LIN{ E6POS: X 741.7167, Y -17.0940, Z -126.0150, A 0, B 90, C 0, E1 0, E2 0, E3 0, E4 0 } C_DIS
LIN{ E6POS: X 740.7177, Y -17.1387, Z -126.0150, A 0, B 90, C 0, E1 0, E2 0, E3 0, E4 0 } C_DIS
LIN{ E6POS: X 739.8800, Y -17.1763, Z -126.0150, A 0, B 90, C 0, E1 0, E2 0, E3 0, E4 0 } C_DIS
LIN{ E6POS: X 739.6024, Y -17.2342, Z -126.0150, A 0, B 90, C 0, E1 0, E2 0, E3 0, E4 0 } C_DIS
LIN{ E6POS: X 738.6175, Y -17.4075, Z -126.0150, A 0, B 90, C 0, E1 0, E2 0, E3 0, E4 0 } C_DIS
LIN{ E6POS: X 737.6326, Y -17.5807, Z -126.0150, A 0, B 90, C 0, E1 0, E2 0, E3 0, E4 0 } C_DIS
LIN{ E6POS: X 736.6477, Y -17.7539, Z -126.0150, A 0, B 90, C 0, E1 0, E2 0, E3 0, E4 0 } C_DIS
LIN{ E6POS: X 736.0951, Y -17.8511, Z -126.0150, A 0, B 90, C 0, E1 0, E2 0, E3 0, E4 0 } C_DIS
LIN{ E6POS: X 736.0012, Y -17.9380, Z -126.0150, A 0, B 90, C 0, E1 0, E2 0, E3 0, E4 0 } C_DIS
LIN{ E6POS: X 735.2228, Y -18.5657, Z -126.0150, A 0, B 90, C 0, E1 0, E2 0, E3 0, E4 0 } C_DIS
LIN{ E6POS: X 734.8225, Y -18.8885, Z -126.0150, A 0, B 90, C 0, E1 0, E2 0, E3 0, E4 0 } C_DIS
LIN{ E6POS: X 735.4953, Y -19.6283, Z -126.0150, A 0, B 90, C 0, E1 0, E2 0, E3 0, E4 0 } C_DIS
LIN{ E6POS: X 735.9742, Y -20.1550, Z -126.0150, A 0, B 90, C 0, E1 0, E2 0, E3 0, E4 0 } C_DIS
LIN{ E6POS: X 736.0644, Y -20.2679, Z -126.0150, A 0, B 90, C 0, E1 0, E2 0, E3 0, E4 0 } C_DIS
LIN{ E6POS: X 736.9769, Y -20.6771, Z -126.0150, A 0, B 90, C 0, E1 0, E2 0, E3 0, E4 0 } C_DIS
LIN{ E6POS: X 737.8893, Y -21.0862, Z -126.0150, A 0, B 90, C 0, E1 0, E2 0, E3 0, E4 0 } C_DIS
LIN{ E6POS: X 738.8018, Y -21.4953, Z -126.0150, A 0, B 90, C 0, E1 0, E2 0, E3 0, E4 0 } C_DIS
LIN{ E6POS: X 739.5476, Y -21.8297, Z -126.0150, A 0, B 90, C 0, E1 0, E2 0, E3 0, E4 0 } C_DIS
LIN{ E6POS: X 739.8221, Y -21.9661, Z -126.0150, A 0, B 90, C 0, E1 0, E2 0, E3 0, E4 0 } C_DIS
LIN{ E6POS: X 740.7757, Y -22.2672, Z -126.0150, A 0, B 90, C 0, E1 0, E2 0, E3 0, E4 0 } C_DIS
LIN{ E6POS: X 741.7293, Y -22.5683, Z -126.0150, A 0, B 90, C 0, E1 0, E2 0, E3 0, E4 0 } C_DIS
LIN{ E6POS: X 742.6829, Y -22.8694, Z -126.0150, A 0, B 90, C 0, E1 0, E2 0, E3 0, E4 0 } C_DIS
LIN{ E6POS: X 743.6365, Y -23.1705, Z -126.0150, A 0, B 90, C 0, E1 0, E2 0, E3 0, E4 0 } C_DIS
LIN{ E6POS: X 744.5901, Y -23.4716, Z -126.0150, A 0, B 90, C 0, E1 0, E2 0, E3 0, E4 0 } C_DIS
LIN{ E6POS: X 745.5437, Y -23.7727, Z -126.0150, A 0, B 90, C 0, E1 0, E2 0, E3 0, E4 0 } C_DIS
LIN{ E6POS: X 745.6394, Y -23.8029, Z -126.0150, A 0, B 90, C 0, E1 0, E2 0, E3 0, E4 0 } C_DIS
LIN{ E6POS: X 746.0988, Y -23.9598, Z -126.0150, A 0, B 90, C 0, E1 0, E2 0, E3 0, E4 0 } C_DIS
LIN{ E6POS: X 747.0681, Y -24.2056, Z -126.0150, A 0, B 90, C 0, E1 0, E2 0, E3 0, E4 0 } C_DIS
LIN{ E6POS: X 748.0375, Y -24.4513, Z -126.0150, A 0, B 90, C 0, E1 0, E2 0, E3 0, E4 0 } C_DIS
LIN{ E6POS: X 749.0068, Y -24.6971, Z -126.0150, A 0, B 90, C 0, E1 0, E2 0, E3 0, E4 0 } C_DIS
LIN{ E6POS: X 749.9761, Y -24.9428, Z -126.0150, A 0, B 90, C 0, E1 0, E2 0, E3 0, E4 0 } C_DIS
LIN{ E6POS: X 750.9455, Y -25.1886, Z -126.0150, A 0, B 90, C 0, E1 0, E2 0, E3 0, E4 0 } C_DIS
LIN{ E6POS: X 751.9148, Y -25.4344, Z -126.0150, A 0, B 90, C 0, E1 0, E2 0, E3 0, E4 0 } C_DIS
LIN{ E6POS: X 752.8841, Y -25.6801, Z -126.0150, A 0, B 90, C 0, E1 0, E2 0, E3 0, E4 0 } C_DIS
LIN{ E6POS: X 753.3483, Y -25.7978, Z -126.0150, A 0, B 90, C 0, E1 0, E2 0, E3 0, E4 0 } C_DIS
LIN{ E6POS: X 753.9231, Y -25.9528, Z -126.0150, A 0, B 90, C 0, E1 0, E2 0, E3 0, E4 0 } C_DIS
LIN{ E6POS: X 754.9035, Y -26.1500, Z -126.0150, A 0, B 90, C 0, E1 0, E2 0, E3 0, E4 0 } C_DIS
LIN{ E6POS: X 755.8838, Y -26.3472, Z -126.0150, A 0, B 90, C 0, E1 0, E2 0, E3 0, E4 0 } C_DIS
LIN{ E6POS: X 756.8642, Y -26.5444, Z -126.0150, A 0, B 90, C 0, E1 0, E2 0, E3 0, E4 0 } C_DIS
LIN{ E6POS: X 757.8446, Y -26.7416, Z -126.0150, A 0, B 90, C 0, E1 0, E2 0, E3 0, E4 0 } C_DIS
LIN{ E6POS: X 758.8249, Y -26.9388, Z -126.0150, A 0, B 90, C 0, E1 0, E2 0, E3 0, E4 0 } C_DIS
LIN{ E6POS: X 759.8053, Y -27.1360, Z -126.0150, A 0, B 90, C 0, E1 0, E2 0, E3 0, E4 0 } C_DIS
LIN{ E6POS: X 760.7857, Y -27.3332, Z -126.0150, A 0, B 90, C 0, E1 0, E2 0, E3 0, E4 0 } C_DIS
LIN{ E6POS: X 761.7005, Y -27.5172, Z -126.0150, A 0, B 90, C 0, E1 0, E2 0, E3 0, E4 0 } C_DIS
LIN{ E6POS: X 762.3215, Y -27.6477, Z -126.0150, A 0, B 90, C 0, E1 0, E2 0, E3 0, E4 0 } C_DIS
LIN{ E6POS: X 763.3122, Y -27.7837, Z -126.0150, A 0, B 90, C 0, E1 0, E2 0, E3 0, E4 0 } C_DIS
LIN{ E6POS: X 764.3029, Y -27.9196, Z -126.0150, A 0, B 90, C 0, E1 0, E2 0, E3 0, E4 0 } C_DIS
LIN{ E6POS: X 765.2937, Y -28.0556, Z -126.0150, A 0, B 90, C 0, E1 0, E2 0, E3 0, E4 0 } C_DIS
LIN{ E6POS: X 766.2844, Y -28.1916, Z -126.0150, A 0, B 90, C 0, E1 0, E2 0, E3 0, E4 0 } C_DIS
LIN{ E6POS: X 767.2751, Y -28.3276, Z -126.0150, A 0, B 90, C 0, E1 0, E2 0, E3 0, E4 0 } C_DIS
LIN{ E6POS: X 768.2658, Y -28.4636, Z -126.0150, A 0, B 90, C 0, E1 0, E2 0, E3 0, E4 0 } C_DIS
LIN{ E6POS: X 769.2565, Y -28.5995, Z -126.0150, A 0, B 90, C 0, E1 0, E2 0, E3 0, E4 0 } C_DIS
LIN{ E6POS: X 769.7261, Y -28.6640, Z -126.0150, A 0, B 90, C 0, E1 0, E2 0, E3 0, E4 0 } C_DIS
LIN{ E6POS: X 770.3238, Y -28.7475, Z -126.0150, A 0, B 90, C 0, E1 0, E2 0, E3 0, E4 0 } C_DIS
LIN{ E6POS: X 771.3233, Y -28.7792, Z -126.0150, A 0, B 90, C 0, E1 0, E2 0, E3 0, E4 0 } C_DIS
LIN{ E6POS: X 772.3228, Y -28.8109, Z -126.0150, A 0, B 90, C 0, E1 0, E2 0, E3 0, E4 0 } C_DIS
LIN{ E6POS: X 773.3223, Y -28.8426, Z -126.0150, A 0, B 90, C 0, E1 0, E2 0, E3 0, E4 0 } C_DIS
LIN{ E6POS: X 774.3218, Y -28.8743, Z -126.0150, A 0, B 90, C 0, E1 0, E2 0, E3 0, E4 0 } C_DIS
LIN{ E6POS: X 775.3213, Y -28.9060, Z -126.0150, A 0, B 90, C 0, E1 0, E2 0, E3 0, E4 0 } C_DIS
LIN{ E6POS: X 776.3208, Y -28.9377, Z -126.0150, A 0, B 90, C 0, E1 0, E2 0, E3 0, E4 0 } C_DIS
LIN{ E6POS: X 776.4510, Y -28.9418, Z -126.0150, A 0, B 90, C 0, E1 0, E2 0, E3 0, E4 0 } C_DIS
LIN{ E6POS: X 776.9561, Y -28.9557, Z -126.0150, A 0, B 90, C 0, E1 0, E2 0, E3 0, E4 0 } C_DIS
LIN{ E6POS: X 777.9387, Y -29.1413, Z -126.0150, A 0, B 90, C 0, E1 0, E2 0, E3 0, E4 0 } C_DIS
LIN{ E6POS: X 778.9214, Y -29.3269, Z -126.0150, A 0, B 90, C 0, E1 0, E2 0, E3 0, E4 0 } C_DIS
LIN{ E6POS: X 779.9040, Y -29.5125, Z -126.0150, A 0, B 90, C 0, E1 0, E2 0, E3 0, E4 0 } C_DIS
LIN{ E6POS: X 780.8866, Y -29.6981, Z -126.0150, A 0, B 90, C 0, E1 0, E2 0, E3 0, E4 0 } C_DIS
LIN{ E6POS: X 781.5842, Y -29.8299, Z -126.0150, A 0, B 90, C 0, E1 0, E2 0, E3 0, E4 0 } C_DIS
LIN{ E6POS: X 781.9729, Y -29.9044, Z -126.0150, A 0, B 90, C 0, E1 0, E2 0, E3 0, E4 0 } C_DIS
LIN{ E6POS: X 782.6620, Y -30.6291, Z -126.0150, A 0, B 90, C 0, E1 0, E2 0, E3 0, E4 0 } C_DIS
LIN{ E6POS: X 783.3511, Y -31.3537, Z -126.0150, A 0, B 90, C 0, E1 0, E2 0, E3 0, E4 0 } C_DIS
LIN{ E6POS: X 784.0403, Y -32.0783, Z -126.0150, A 0, B 90, C 0, E1 0, E2 0, E3 0, E4 0 } C_DIS
LIN{ E6POS: X 784.7294, Y -32.8030, Z -126.0150, A 0, B 90, C 0, E1 0, E2 0, E3 0, E4 0 } C_DIS
LIN{ E6POS: X 784.8800, Y -32.9613, Z -126.0150, A 0, B 90, C 0, E1 0, E2 0, E3 0, E4 0 } C_DIS
LIN{ E6POS: X 785.1281, Y -33.2266, Z -126.0150, A 0, B 90, C 0, E1 0, E2 0, E3 0, E4 0 } C_DIS
LIN{ E6POS: X 785.2695, Y -34.2166, Z -126.0150, A 0, B 90, C 0, E1 0, E2 0, E3 0, E4 0 } C_DIS
LIN{ E6POS: X 785.4109, Y -35.2065, Z -126.0150, A 0, B 90, C 0, E1 0, E2 0, E3 0, E4 0 } C_DIS
LIN{ E6POS: X 785.5523, Y -36.1965, Z -126.0150, A 0, B 90, C 0, E1 0, E2 0, E3 0, E4 0 } C_DIS
LIN{ E6POS: X 785.6937, Y -37.1864, Z -126.0150, A 0, B 90, C 0, E1 0, E2 0, E3 0, E4 0 } C_DIS
LIN{ E6POS: X 785.8351, Y -38.1764, Z -126.0150, A 0, B 90, C 0, E1 0, E2 0, E3 0, E4 0 } C_DIS
LIN{ E6POS: X 785.9765, Y -39.1663, Z -126.0150, A 0, B 90, C 0, E1 0, E2 0, E3 0, E4 0 } C_DIS
LIN{ E6POS: X 786.0909, Y -39.9674, Z -126.0150, A 0, B 90, C 0, E1 0, E2 0, E3 0, E4 0 } C_DIS
LIN{ E6POS: X 786.1747, Y -40.5536, Z -126.0150, A 0, B 90, C 0, E1 0, E2 0, E3 0, E4 0 } C_DIS
LIN{ E6POS: X 786.0743, Y -41.5485, Z -126.0150, A 0, B 90, C 0, E1 0, E2 0, E3 0, E4 0 } C_DIS
LIN{ E6POS: X 785.9740, Y -42.5435, Z -126.0150, A 0, B 90, C 0, E1 0, E2 0, E3 0, E4 0 } C_DIS
LIN{ E6POS: X 785.8737, Y -43.5384, Z -126.0150, A 0, B 90, C 0, E1 0, E2 0, E3 0, E4 0 } C_DIS
LIN{ E6POS: X 785.7734, Y -44.5334, Z -126.0150, A 0, B 90, C 0, E1 0, E2 0, E3 0, E4 0 } C_DIS
LIN{ E6POS: X 785.6731, Y -45.5283, Z -126.0150, A 0, B 90, C 0, E1 0, E2 0, E3 0, E4 0 } C_DIS
LIN{ E6POS: X 785.5728, Y -46.5233, Z -126.0150, A 0, B 90, C 0, E1 0, E2 0, E3 0, E4 0 } C_DIS
LIN{ E6POS: X 785.4725, Y -47.5183, Z -126.0150, A 0, B 90, C 0, E1 0, E2 0, E3 0, E4 0 } C_DIS
LIN{ E6POS: X 785.3721, Y -48.5132, Z -126.0150, A 0, B 90, C 0, E1 0, E2 0, E3 0, E4 0 } C_DIS
LIN{ E6POS: X 785.2718, Y -49.5082, Z -126.0150, A 0, B 90, C 0, E1 0, E2 0, E3 0, E4 0 } C_DIS
LIN{ E6POS: X 785.1715, Y -50.5031, Z -126.0150, A 0, B 90, C 0, E1 0, E2 0, E3 0, E4 0 } C_DIS
LIN{ E6POS: X 785.0712, Y -51.4981, Z -126.0150, A 0, B 90, C 0, E1 0, E2 0, E3 0, E4 0 } C_DIS
LIN{ E6POS: X 784.9721, Y -52.4813, Z -126.0150, A 0, B 90, C 0, E1 0, E2 0, E3 0, E4 0 } C_DIS
LIN{ E6POS: X 784.8718, Y -53.4762, Z -126.0150, A 0, B 90, C 0, E1 0, E2 0, E3 0, E4 0 } C_DIS
LIN{ E6POS: X 784.8675, Y -53.5185, Z -126.0150, A 0, B 90, C 0, E1 0, E2 0, E3 0, E4 0 } C_DIS
LIN{ E6POS: X 784.6915, Y -54.5029, Z -126.0150, A 0, B 90, C 0, E1 0, E2 0, E3 0, E4 0 } C_DIS
LIN{ E6POS: X 784.5156, Y -55.4873, Z -126.0150, A 0, B 90, C 0, E1 0, E2 0, E3 0, E4 0 } C_DIS
LIN{ E6POS: X 784.3396, Y -56.4717, Z -126.0150, A 0, B 90, C 0, E1 0, E2 0, E3 0, E4 0 } C_DIS
LIN{ E6POS: X 784.1637, Y -57.4560, Z -126.0150, A 0, B 90, C 0, E1 0, E2 0, E3 0, E4 0 } C_DIS
LIN{ E6POS: X 783.9877, Y -58.4404, Z -126.0150, A 0, B 90, C 0, E1 0, E2 0, E3 0, E4 0 } C_DIS
LIN{ E6POS: X 783.8118, Y -59.4248, Z -126.0150, A 0, B 90, C 0, E1 0, E2 0, E3 0, E4 0 } C_DIS
LIN{ E6POS: X 783.6358, Y -60.4092, Z -126.0150, A 0, B 90, C 0, E1 0, E2 0, E3 0, E4 0 } C_DIS
LIN{ E6POS: X 783.4599, Y -61.3936, Z -126.0150, A 0, B 90, C 0, E1 0, E2 0, E3 0, E4 0 } C_DIS
LIN{ E6POS: X 783.2839, Y -62.3780, Z -126.0150, A 0, B 90, C 0, E1 0, E2 0, E3 0, E4 0 } C_DIS
LIN{ E6POS: X 783.1080, Y -63.3624, Z -126.0150, A 0, B 90, C 0, E1 0, E2 0, E3 0, E4 0 } C_DIS
LIN{ E6POS: X 782.9320, Y -64.3468, Z -126.0150, A 0, B 90, C 0, E1 0, E2 0, E3 0, E4 0 } C_DIS
LIN{ E6POS: X 782.7561, Y -65.3312, Z -126.0150, A 0, B 90, C 0, E1 0, E2 0, E3 0, E4 0 } C_DIS
LIN{ E6POS: X 782.5801, Y -66.3156, Z -126.0150, A 0, B 90, C 0, E1 0, E2 0, E3 0, E4 0 } C_DIS
LIN{ E6POS: X 782.4042, Y -67.3000, Z -126.0150, A 0, B 90, C 0, E1 0, E2 0, E3 0, E4 0 } C_DIS
LIN{ E6POS: X 782.2282, Y -68.2844, Z -126.0150, A 0, B 90, C 0, E1 0, E2 0, E3 0, E4 0 } C_DIS
LIN{ E6POS: X 782.0523, Y -69.2688, Z -126.0150, A 0, B 90, C 0, E1 0, E2 0, E3 0, E4 0 } C_DIS
LIN{ E6POS: X 782.0402, Y -69.3364, Z -126.0150, A 0, B 90, C 0, E1 0, E2 0, E3 0, E4 0 } C_DIS
LIN{ E6POS: X 781.8642, Y -70.3208, Z -126.0150, A 0, B 90, C 0, E1 0, E2 0, E3 0, E4 0 } C_DIS
LIN{ E6POS: X 781.7943, Y -70.7119, Z -126.0150, A 0, B 90, C 0, E1 0, E2 0, E3 0, E4 0 } C_DIS
LIN{ E6POS: X 781.5865, Y -71.6900, Z -126.0150, A 0, B 90, C 0, E1 0, E2 0, E3 0, E4 0 } C_DIS
LIN{ E6POS: X 781.3787, Y -72.6682, Z -126.0150, A 0, B 90, C 0, E1 0, E2 0, E3 0, E4 0 } C_DIS
LIN{ E6POS: X 781.1709, Y -73.6464, Z -126.0150, A 0, B 90, C 0, E1 0, E2 0, E3 0, E4 0 } C_DIS
LIN{ E6POS: X 780.9631, Y -74.6245, Z -126.0150, A 0, B 90, C 0, E1 0, E2 0, E3 0, E4 0 } C_DIS
LIN{ E6POS: X 780.7553, Y -75.6027, Z -126.0150, A 0, B 90, C 0, E1 0, E2 0, E3 0, E4 0 } C_DIS
LIN{ E6POS: X 780.5475, Y -76.5809, Z -126.0150, A 0, B 90, C 0, E1 0, E2 0, E3 0, E4 0 } C_DIS
LIN{ E6POS: X 780.3397, Y -77.5590, Z -126.0150, A 0, B 90, C 0, E1 0, E2 0, E3 0, E4 0 } C_DIS
LIN{ E6POS: X 780.1319, Y -78.5372, Z -126.0150, A 0, B 90, C 0, E1 0, E2 0, E3 0, E4 0 } C_DIS
LIN{ E6POS: X 779.9241, Y -79.5154, Z -126.0150, A 0, B 90, C 0, E1 0, E2 0, E3 0, E4 0 } C_DIS
LIN{ E6POS: X 779.7163, Y -80.4936, Z -126.0150, A 0, B 90, C 0, E1 0, E2 0, E3 0, E4 0 } C_DIS
LIN{ E6POS: X 779.5085, Y -81.4717, Z -126.0150, A 0, B 90, C 0, E1 0, E2 0, E3 0, E4 0 } C_DIS
LIN{ E6POS: X 779.3007, Y -82.4499, Z -126.0150, A 0, B 90, C 0, E1 0, E2 0, E3 0, E4 0 } C_DIS
LIN{ E6POS: X 779.0929, Y -83.4281, Z -126.0150, A 0, B 90, C 0, E1 0, E2 0, E3 0, E4 0 } C_DIS
LIN{ E6POS: X 778.8851, Y -84.4062, Z -126.0150, A 0, B 90, C 0, E1 0, E2 0, E3 0, E4 0 } C_DIS
LIN{ E6POS: X 778.6773, Y -85.3844, Z -126.0150, A 0, B 90, C 0, E1 0, E2 0, E3 0, E4 0 } C_DIS
LIN{ E6POS: X 778.4695, Y -86.3626, Z -126.0150, A 0, B 90, C 0, E1 0, E2 0, E3 0, E4 0 } C_DIS
LIN{ E6POS: X 778.2617, Y -87.3408, Z -126.0150, A 0, B 90, C 0, E1 0, E2 0, E3 0, E4 0 } C_DIS
LIN{ E6POS: X 778.0539, Y -88.3189, Z -126.0150, A 0, B 90, C 0, E1 0, E2 0, E3 0, E4 0 } C_DIS
LIN{ E6POS: X 777.8830, Y -89.1233, Z -126.0150, A 0, B 90, C 0, E1 0, E2 0, E3 0, E4 0 } C_DIS
LIN{ E6POS: X 777.6752, Y -90.1015, Z -126.0150, A 0, B 90, C 0, E1 0, E2 0, E3 0, E4 0 } C_DIS
LIN{ E6POS: X 777.5429, Y -90.7243, Z -126.0150, A 0, B 90, C 0, E1 0, E2 0, E3 0, E4 0 } C_DIS
LIN{ E6POS: X 777.3226, Y -91.6997, Z -126.0150, A 0, B 90, C 0, E1 0, E2 0, E3 0, E4 0 } C_DIS
LIN{ E6POS: X 777.1022, Y -92.6751, Z -126.0150, A 0, B 90, C 0, E1 0, E2 0, E3 0, E4 0 } C_DIS
LIN{ E6POS: X 776.8819, Y -93.6506, Z -126.0150, A 0, B 90, C 0, E1 0, E2 0, E3 0, E4 0 } C_DIS
LIN{ E6POS: X 776.6615, Y -94.6260, Z -126.0150, A 0, B 90, C 0, E1 0, E2 0, E3 0, E4 0 } C_DIS
LIN{ E6POS: X 776.4412, Y -95.6014, Z -126.0150, A 0, B 90, C 0, E1 0, E2 0, E3 0, E4 0 } C_DIS
LIN{ E6POS: X 776.2208, Y -96.5768, Z -126.0150, A 0, B 90, C 0, E1 0, E2 0, E3 0, E4 0 } C_DIS
LIN{ E6POS: X 776.0005, Y -97.5522, Z -126.0150, A 0, B 90, C 0, E1 0, E2 0, E3 0, E4 0 } C_DIS
LIN{ E6POS: X 775.7802, Y -98.5277, Z -126.0150, A 0, B 90, C 0, E1 0, E2 0, E3 0, E4 0 } C_DIS
LIN{ E6POS: X 775.5598, Y -99.5031, Z -126.0150, A 0, B 90, C 0, E1 0, E2 0, E3 0, E4 0 } C_DIS
LIN{ E6POS: X 775.3395, Y -100.4785, Z -126.0150, A 0, B 90, C 0, E1 0, E2 0, E3 0, E4 0 } C_DIS
LIN{ E6POS: X 775.1191, Y -101.4539, Z -126.0150, A 0, B 90, C 0, E1 0, E2 0, E3 0, E4 0 } C_DIS
LIN{ E6POS: X 774.8988, Y -102.4294, Z -126.0150, A 0, B 90, C 0, E1 0, E2 0, E3 0, E4 0 } C_DIS
LIN{ E6POS: X 774.6784, Y -103.4048, Z -126.0150, A 0, B 90, C 0, E1 0, E2 0, E3 0, E4 0 } C_DIS
LIN{ E6POS: X 774.4581, Y -104.3802, Z -126.0150, A 0, B 90, C 0, E1 0, E2 0, E3 0, E4 0 } C_DIS
LIN{ E6POS: X 774.2377, Y -105.3556, Z -126.0150, A 0, B 90, C 0, E1 0, E2 0, E3 0, E4 0 } C_DIS
LIN{ E6POS: X 774.0174, Y -106.3310, Z -126.0150, A 0, B 90, C 0, E1 0, E2 0, E3 0, E4 0 } C_DIS
LIN{ E6POS: X 773.7970, Y -107.3065, Z -126.0150, A 0, B 90, C 0, E1 0, E2 0, E3 0, E4 0 } C_DIS
LIN{ E6POS: X 773.5767, Y -108.2819, Z -126.0150, A 0, B 90, C 0, E1 0, E2 0, E3 0, E4 0 } C_DIS
LIN{ E6POS: X 773.3564, Y -109.2573, Z -126.0150, A 0, B 90, C 0, E1 0, E2 0, E3 0, E4 0 } C_DIS
LIN{ E6POS: X 773.1360, Y -110.2327, Z -126.0150, A 0, B 90, C 0, E1 0, E2 0, E3 0, E4 0 } C_DIS
LIN{ E6POS: X 773.0909, Y -110.4324, Z -126.0150, A 0, B 90, C 0, E1 0, E2 0, E3 0, E4 0 } C_DIS
LIN{ E6POS: X 772.8706, Y -111.4079, Z -126.0150, A 0, B 90, C 0, E1 0, E2 0, E3 0, E4 0 } C_DIS
LIN{ E6POS: X 772.7038, Y -112.1462, Z -126.0150, A 0, B 90, C 0, E1 0, E2 0, E3 0, E4 0 } C_DIS
LIN{ E6POS: X 772.0412, Y -111.3972, Z -126.0150, A 0, B 90, C 0, E1 0, E2 0, E3 0, E4 0 } C_DIS
LIN{ E6POS: X 771.3787, Y -110.6481, Z -126.0150, A 0, B 90, C 0, E1 0, E2 0, E3 0, E4 0 } C_DIS
LIN{ E6POS: X 770.7162, Y -109.8991, Z -126.0150, A 0, B 90, C 0, E1 0, E2 0, E3 0, E4 0 } C_DIS
LIN{ E6POS: X 770.2453, Y -109.3667, Z -126.0150, A 0, B 90, C 0, E1 0, E2 0, E3 0, E4 0 } C_DIS
LIN{ E6POS: X 770.0315, Y -109.1250, Z -126.0150, A 0, B 90, C 0, E1 0, E2 0, E3 0, E4 0 } C_DIS
LIN{ E6POS: X 769.2905, Y -108.4535, Z -126.0150, A 0, B 90, C 0, E1 0, E2 0, E3 0, E4 0 } C_DIS
LIN{ E6POS: X 768.5495, Y -107.7819, Z -126.0150, A 0, B 90, C 0, E1 0, E2 0, E3 0, E4 0 } C_DIS
LIN{ E6POS: X 767.8086, Y -107.1104, Z -126.0150, A 0, B 90, C 0, E1 0, E2 0, E3 0, E4 0 } C_DIS
LIN{ E6POS: X 767.0676, Y -106.4389, Z -126.0150, A 0, B 90, C 0, E1 0, E2 0, E3 0, E4 0 } C_DIS
LIN{ E6POS: X 766.8332, Y -106.2265, Z -126.0150, A 0, B 90, C 0, E1 0, E2 0, E3 0, E4 0 } C_DIS
LIN{ E6POS: X 766.5571, Y -105.9757, Z -126.0150, A 0, B 90, C 0, E1 0, E2 0, E3 0, E4 0 } C_DIS
LIN{ E6POS: X 766.1563, Y -105.7065, Z -126.0150, A 0, B 90, C 0, E1 0, E2 0, E3 0, E4 0 } C_DIS
LIN{ E6POS: X 765.3256, Y -105.1498, Z -126.0150, A 0, B 90, C 0, E1 0, E2 0, E3 0, E4 0 } C_DIS
LIN{ E6POS: X 764.4949, Y -104.5931, Z -126.0150, A 0, B 90, C 0, E1 0, E2 0, E3 0, E4 0 } C_DIS
LIN{ E6POS: X 763.6642, Y -104.0363, Z -126.0150, A 0, B 90, C 0, E1 0, E2 0, E3 0, E4 0 } C_DIS
LIN{ E6POS: X 762.8335, Y -103.4796, Z -126.0150, A 0, B 90, C 0, E1 0, E2 0, E3 0, E4 0 } C_DIS
LIN{ E6POS: X 762.0028, Y -102.9229, Z -126.0150, A 0, B 90, C 0, E1 0, E2 0, E3 0, E4 0 } C_DIS
LIN{ E6POS: X 761.4803, Y -102.5727, Z -126.0150, A 0, B 90, C 0, E1 0, E2 0, E3 0, E4 0 } C_DIS
LIN{ E6POS: X 760.8926, Y -102.2760, Z -126.0150, A 0, B 90, C 0, E1 0, E2 0, E3 0, E4 0 } C_DIS
LIN{ E6POS: X 760.0004, Y -101.8244, Z -126.0150, A 0, B 90, C 0, E1 0, E2 0, E3 0, E4 0 } C_DIS
LIN{ E6POS: X 759.1082, Y -101.3728, Z -126.0150, A 0, B 90, C 0, E1 0, E2 0, E3 0, E4 0 } C_DIS
LIN{ E6POS: X 758.2159, Y -100.9213, Z -126.0150, A 0, B 90, C 0, E1 0, E2 0, E3 0, E4 0 } C_DIS
LIN{ E6POS: X 757.3237, Y -100.4697, Z -126.0150, A 0, B 90, C 0, E1 0, E2 0, E3 0, E4 0 } C_DIS
LIN{ E6POS: X 756.4315, Y -100.0181, Z -126.0150, A 0, B 90, C 0, E1 0, E2 0, E3 0, E4 0 } C_DIS
LIN{ E6POS: X 755.5392, Y -99.5665, Z -126.0150, A 0, B 90, C 0, E1 0, E2 0, E3 0, E4 0 } C_DIS
LIN{ E6POS: X 754.6470, Y -99.1150, Z -126.0150, A 0, B 90, C 0, E1 0, E2 0, E3 0, E4 0 } C_DIS
LIN{ E6POS: X 753.9986, Y -98.7868, Z -126.0150, A 0, B 90, C 0, E1 0, E2 0, E3 0, E4 0 } C_DIS
LIN{ E6POS: X 753.1615, Y -98.4535, Z -126.0150, A 0, B 90, C 0, E1 0, E2 0, E3 0, E4 0 } C_DIS
LIN{ E6POS: X 752.2338, Y -98.0803, Z -126.0150, A 0, B 90, C 0, E1 0, E2 0, E3 0, E4 0 } C_DIS
LIN{ E6POS: X 751.3060, Y -97.7070, Z -126.0150, A 0, B 90, C 0, E1 0, E2 0, E3 0, E4 0 } C_DIS
LIN{ E6POS: X 750.3783, Y -97.3338, Z -126.0150, A 0, B 90, C 0, E1 0, E2 0, E3 0, E4 0 } C_DIS
LIN{ E6POS: X 749.4506, Y -96.9605, Z -126.0150, A 0, B 90, C 0, E1 0, E2 0, E3 0, E4 0 } C_DIS
LIN{ E6POS: X 748.5228, Y -96.5873, Z -126.0150, A 0, B 90, C 0, E1 0, E2 0, E3 0, E4 0 } C_DIS
LIN{ E6POS: X 747.5951, Y -96.2140, Z -126.0150, A 0, B 90, C 0, E1 0, E2 0, E3 0, E4 0 } C_DIS
LIN{ E6POS: X 746.6674, Y -95.8408, Z -126.0150, A 0, B 90, C 0, E1 0, E2 0, E3 0, E4 0 } C_DIS
LIN{ E6POS: X 745.7396, Y -95.4675, Z -126.0150, A 0, B 90, C 0, E1 0, E2 0, E3 0, E4 0 } C_DIS
LIN{ E6POS: X 744.8119, Y -95.0943, Z -126.0150, A 0, B 90, C 0, E1 0, E2 0, E3 0, E4 0 } C_DIS
LIN{ E6POS: X 743.8842, Y -94.7210, Z -126.0150, A 0, B 90, C 0, E1 0, E2 0, E3 0, E4 0 } C_DIS
LIN{ E6POS: X 743.3112, Y -94.4905, Z -126.0150, A 0, B 90, C 0, E1 0, E2 0, E3 0, E4 0 } C_DIS
LIN{ E6POS: X 742.3695, Y -94.1539, Z -126.0150, A 0, B 90, C 0, E1 0, E2 0, E3 0, E4 0 } C_DIS
LIN{ E6POS: X 742.3638, Y -94.1519, Z -126.0150, A 0, B 90, C 0, E1 0, E2 0, E3 0, E4 0 } C_DIS
LIN{ E6POS: X 741.4234, Y -93.8116, Z -126.0150, A 0, B 90, C 0, E1 0, E2 0, E3 0, E4 0 } C_DIS
LIN{ E6POS: X 740.4831, Y -93.4714, Z -126.0150, A 0, B 90, C 0, E1 0, E2 0, E3 0, E4 0 } C_DIS
LIN{ E6POS: X 739.5428, Y -93.1311, Z -126.0150, A 0, B 90, C 0, E1 0, E2 0, E3 0, E4 0 } C_DIS
LIN{ E6POS: X 738.6024, Y -92.7908, Z -126.0150, A 0, B 90, C 0, E1 0, E2 0, E3 0, E4 0 } C_DIS
LIN{ E6POS: X 737.6621, Y -92.4506, Z -126.0150, A 0, B 90, C 0, E1 0, E2 0, E3 0, E4 0 } C_DIS
LIN{ E6POS: X 736.7218, Y -92.1103, Z -126.0150, A 0, B 90, C 0, E1 0, E2 0, E3 0, E4 0 } C_DIS
LIN{ E6POS: X 735.7814, Y -91.7701, Z -126.0150, A 0, B 90, C 0, E1 0, E2 0, E3 0, E4 0 } C_DIS
LIN{ E6POS: X 734.8411, Y -91.4298, Z -126.0150, A 0, B 90, C 0, E1 0, E2 0, E3 0, E4 0 } C_DIS
LIN{ E6POS: X 733.9008, Y -91.0896, Z -126.0150, A 0, B 90, C 0, E1 0, E2 0, E3 0, E4 0 } C_DIS
LIN{ E6POS: X 732.9604, Y -90.7493, Z -126.0150, A 0, B 90, C 0, E1 0, E2 0, E3 0, E4 0 } C_DIS
LIN{ E6POS: X 732.0201, Y -90.4091, Z -126.0150, A 0, B 90, C 0, E1 0, E2 0, E3 0, E4 0 } C_DIS
LIN{ E6POS: X 731.1955, Y -90.1107, Z -126.0150, A 0, B 90, C 0, E1 0, E2 0, E3 0, E4 0 } C_DIS
LIN{ E6POS: X 730.2766, Y -89.7980, Z -126.0150, A 0, B 90, C 0, E1 0, E2 0, E3 0, E4 0 } C_DIS
LIN{ E6POS: X 729.3309, Y -89.4731, Z -126.0150, A 0, B 90, C 0, E1 0, E2 0, E3 0, E4 0 } C_DIS
LIN{ E6POS: X 728.3851, Y -89.1482, Z -126.0150, A 0, B 90, C 0, E1 0, E2 0, E3 0, E4 0 } C_DIS
LIN{ E6POS: X 727.4394, Y -88.8233, Z -126.0150, A 0, B 90, C 0, E1 0, E2 0, E3 0, E4 0 } C_DIS
LIN{ E6POS: X 726.4936, Y -88.4984, Z -126.0150, A 0, B 90, C 0, E1 0, E2 0, E3 0, E4 0 } C_DIS
LIN{ E6POS: X 725.5479, Y -88.1735, Z -126.0150, A 0, B 90, C 0, E1 0, E2 0, E3 0, E4 0 } C_DIS
LIN{ E6POS: X 724.6021, Y -87.8486, Z -126.0150, A 0, B 90, C 0, E1 0, E2 0, E3 0, E4 0 } C_DIS
LIN{ E6POS: X 723.6564, Y -87.5237, Z -126.0150, A 0, B 90, C 0, E1 0, E2 0, E3 0, E4 0 } C_DIS
LIN{ E6POS: X 722.7106, Y -87.1988, Z -126.0150, A 0, B 90, C 0, E1 0, E2 0, E3 0, E4 0 } C_DIS
LIN{ E6POS: X 721.7649, Y -86.8739, Z -126.0150, A 0, B 90, C 0, E1 0, E2 0, E3 0, E4 0 } C_DIS
LIN{ E6POS: X 720.8191, Y -86.5490, Z -126.0150, A 0, B 90, C 0, E1 0, E2 0, E3 0, E4 0 } C_DIS
LIN{ E6POS: X 719.8734, Y -86.2242, Z -126.0150, A 0, B 90, C 0, E1 0, E2 0, E3 0, E4 0 } C_DIS
LIN{ E6POS: X 719.4295, Y -86.0717, Z -126.0150, A 0, B 90, C 0, E1 0, E2 0, E3 0, E4 0 } C_DIS
LIN{ E6POS: X 718.6780, Y -85.8163, Z -126.0150, A 0, B 90, C 0, E1 0, E2 0, E3 0, E4 0 } C_DIS
LIN{ E6POS: X 717.7311, Y -85.4947, Z -126.0150, A 0, B 90, C 0, E1 0, E2 0, E3 0, E4 0 } C_DIS
LIN{ E6POS: X 716.7842, Y -85.1732, Z -126.0150, A 0, B 90, C 0, E1 0, E2 0, E3 0, E4 0 } C_DIS
LIN{ E6POS: X 715.8373, Y -84.8517, Z -126.0150, A 0, B 90, C 0, E1 0, E2 0, E3 0, E4 0 } C_DIS
LIN{ E6POS: X 714.8904, Y -84.5302, Z -126.0150, A 0, B 90, C 0, E1 0, E2 0, E3 0, E4 0 } C_DIS
LIN{ E6POS: X 713.9435, Y -84.2087, Z -126.0150, A 0, B 90, C 0, E1 0, E2 0, E3 0, E4 0 } C_DIS
LIN{ E6POS: X 712.9966, Y -83.8871, Z -126.0150, A 0, B 90, C 0, E1 0, E2 0, E3 0, E4 0 } C_DIS
LIN{ E6POS: X 712.0497, Y -83.5656, Z -126.0150, A 0, B 90, C 0, E1 0, E2 0, E3 0, E4 0 } C_DIS
LIN{ E6POS: X 711.1028, Y -83.2441, Z -126.0150, A 0, B 90, C 0, E1 0, E2 0, E3 0, E4 0 } C_DIS
LIN{ E6POS: X 710.1559, Y -82.9226, Z -126.0150, A 0, B 90, C 0, E1 0, E2 0, E3 0, E4 0 } C_DIS
LIN{ E6POS: X 709.7916, Y -82.7989, Z -126.0150, A 0, B 90, C 0, E1 0, E2 0, E3 0, E4 0 } C_DIS
LIN{ E6POS: X 709.3465, Y -82.6322, Z -126.0150, A 0, B 90, C 0, E1 0, E2 0, E3 0, E4 0 } C_DIS
LIN{ E6POS: X 708.4062, Y -82.2918, Z -126.0150, A 0, B 90, C 0, E1 0, E2 0, E3 0, E4 0 } C_DIS
LIN{ E6POS: X 707.4659, Y -81.9515, Z -126.0150, A 0, B 90, C 0, E1 0, E2 0, E3 0, E4 0 } C_DIS
LIN{ E6POS: X 706.5256, Y -81.6111, Z -126.0150, A 0, B 90, C 0, E1 0, E2 0, E3 0, E4 0 } C_DIS
LIN{ E6POS: X 705.5853, Y -81.2708, Z -126.0150, A 0, B 90, C 0, E1 0, E2 0, E3 0, E4 0 } C_DIS
LIN{ E6POS: X 704.6450, Y -80.9305, Z -126.0150, A 0, B 90, C 0, E1 0, E2 0, E3 0, E4 0 } C_DIS
LIN{ E6POS: X 704.0586, Y -80.7182, Z -126.0150, A 0, B 90, C 0, E1 0, E2 0, E3 0, E4 0 } C_DIS
LIN{ E6POS: X 703.8433, Y -80.6180, Z -126.0150, A 0, B 90, C 0, E1 0, E2 0, E3 0, E4 0 } C_DIS
LIN{ E6POS: X 702.9212, Y -80.2310, Z -126.0150, A 0, B 90, C 0, E1 0, E2 0, E3 0, E4 0 } C_DIS
LIN{ E6POS: X 701.9991, Y -79.8440, Z -126.0150, A 0, B 90, C 0, E1 0, E2 0, E3 0, E4 0 } C_DIS
LIN{ E6POS: X 701.2543, Y -79.5315, Z -126.0150, A 0, B 90, C 0, E1 0, E2 0, E3 0, E4 0 } C_DIS
LIN{ E6POS: X 701.2019, Y -79.4530, Z -126.0150, A 0, B 90, C 0, E1 0, E2 0, E3 0, E4 0 } C_DIS
LIN{ E6POS: X 700.4916, Y -78.7491, Z -126.0150, A 0, B 90, C 0, E1 0, E2 0, E3 0, E4 0 } C_DIS
LIN{ E6POS: X 700.4879, Y -78.7454, Z -126.0150, A 0, B 90, C 0, E1 0, E2 0, E3 0, E4 0 } C_DIS
LIN{ E6POS: X 700.7255, Y -77.7740, Z -126.0150, A 0, B 90, C 0, E1 0, E2 0, E3 0, E4 0 } C_DIS
LIN{ E6POS: X 700.8261, Y -77.3633, Z -126.0150, A 0, B 90, C 0, E1 0, E2 0, E3 0, E4 0 } C_DIS
LIN{ E6POS: X 700.8626, Y -77.2328, Z -126.0150, A 0, B 90, C 0, E1 0, E2 0, E3 0, E4 0 } C_DIS
LIN{ E6POS: X 701.0928, Y -76.2597, Z -126.0150, A 0, B 90, C 0, E1 0, E2 0, E3 0, E4 0 } C_DIS
LIN{ E6POS: X 701.1686, Y -75.9391, Z -126.0150, A 0, B 90, C 0, E1 0, E2 0, E3 0, E4 0 } C_DIS
LIN{ E6POS: X 701.2004, Y -75.8212, Z -126.0150, A 0, B 90, C 0, E1 0, E2 0, E3 0, E4 0 } C_DIS
LIN{ E6POS: X 701.4360, Y -74.8493, Z -126.0150, A 0, B 90, C 0, E1 0, E2 0, E3 0, E4 0 } C_DIS
LIN{ E6POS: X 701.5128, Y -74.5323, Z -126.0150, A 0, B 90, C 0, E1 0, E2 0, E3 0, E4 0 } C_DIS
LIN{ E6POS: X 701.5447, Y -74.4166, Z -126.0150, A 0, B 90, C 0, E1 0, E2 0, E3 0, E4 0 } C_DIS
LIN{ E6POS: X 701.7895, Y -73.4470, Z -126.0150, A 0, B 90, C 0, E1 0, E2 0, E3 0, E4 0 } C_DIS
LIN{ E6POS: X 701.8681, Y -73.1360, Z -126.0150, A 0, B 90, C 0, E1 0, E2 0, E3 0, E4 0 } C_DIS
LIN{ E6POS: X 701.9001, Y -73.0237, Z -126.0150, A 0, B 90, C 0, E1 0, E2 0, E3 0, E4 0 } C_DIS
LIN{ E6POS: X 702.1561, Y -72.0570, Z -126.0150, A 0, B 90, C 0, E1 0, E2 0, E3 0, E4 0 } C_DIS
LIN{ E6POS: X 702.2370, Y -71.7511, Z -126.0150, A 0, B 90, C 0, E1 0, E2 0, E3 0, E4 0 } C_DIS
LIN{ E6POS: X 702.2693, Y -71.6434, Z -126.0150, A 0, B 90, C 0, E1 0, E2 0, E3 0, E4 0 } C_DIS
LIN{ E6POS: X 702.5295, Y -70.6778, Z -126.0150, A 0, B 90, C 0, E1 0, E2 0, E3 0, E4 0 } C_DIS
LIN{ E6POS: X 702.6134, Y -70.3664, Z -126.0150, A 0, B 90, C 0, E1 0, E2 0, E3 0, E4 0 } C_DIS
LIN{ E6POS: X 702.6454, Y -70.2605, Z -126.0150, A 0, B 90, C 0, E1 0, E2 0, E3 0, E4 0 } C_DIS
LIN{ E6POS: X 702.9019, Y -69.2939, Z -126.0150, A 0, B 90, C 0, E1 0, E2 0, E3 0, E4 0 } C_DIS
LIN{ E6POS: X 702.9891, Y -68.9652, Z -126.0150, A 0, B 90, C 0, E1 0, E2 0, E3 0, E4 0 } C_DIS
LIN{ E6POS: X 703.0207, Y -68.8585, Z -126.0150, A 0, B 90, C 0, E1 0, E2 0, E3 0, E4 0 } C_DIS
LIN{ E6POS: X 703.2656, Y -67.8890, Z -126.0150, A 0, B 90, C 0, E1 0, E2 0, E3 0, E4 0 } C_DIS
LIN{ E6POS: X 703.3563, Y -67.5301, Z -126.0150, A 0, B 90, C 0, E1 0, E2 0, E3 0, E4 0 } C_DIS
LIN{ E6POS: X 703.3872, Y -67.4199, Z -126.0150, A 0, B 90, C 0, E1 0, E2 0, E3 0, E4 0 } C_DIS
LIN{ E6POS: X 703.6144, Y -66.4461, Z -126.0150, A 0, B 90, C 0, E1 0, E2 0, E3 0, E4 0 } C_DIS
LIN{ E6POS: X 703.7083, Y -66.0439, Z -126.0150, A 0, B 90, C 0, E1 0, E2 0, E3 0, E4 0 } C_DIS
LIN{ E6POS: X 703.7380, Y -65.9276, Z -126.0150, A 0, B 90, C 0, E1 0, E2 0, E3 0, E4 0 } C_DIS
LIN{ E6POS: X 703.9521, Y -64.9508, Z -126.0150, A 0, B 90, C 0, E1 0, E2 0, E3 0, E4 0 } C_DIS
LIN{ E6POS: X 704.0426, Y -64.5378, Z -126.0150, A 0, B 90, C 0, E1 0, E2 0, E3 0, E4 0 } C_DIS
LIN{ E6POS: X 704.0713, Y -64.4189, Z -126.0150, A 0, B 90, C 0, E1 0, E2 0, E3 0, E4 0 } C_DIS
LIN{ E6POS: X 704.2767, Y -63.4402, Z -126.0150, A 0, B 90, C 0, E1 0, E2 0, E3 0, E4 0 } C_DIS
LIN{ E6POS: X 704.3591, Y -63.0477, Z -126.0150, A 0, B 90, C 0, E1 0, E2 0, E3 0, E4 0 } C_DIS
LIN{ E6POS: X 704.3867, Y -62.9296, Z -126.0150, A 0, B 90, C 0, E1 0, E2 0, E3 0, E4 0 } C_DIS
LIN{ E6POS: X 704.5872, Y -61.9499, Z -126.0150, A 0, B 90, C 0, E1 0, E2 0, E3 0, E4 0 } C_DIS
LIN{ E6POS: X 704.6565, Y -61.6112, Z -126.0150, A 0, B 90, C 0, E1 0, E2 0, E3 0, E4 0 } C_DIS
LIN{ E6POS: X 704.6831, Y -61.4973, Z -126.0150, A 0, B 90, C 0, E1 0, E2 0, E3 0, E4 0 } C_DIS
LIN{ E6POS: X 704.8829, Y -60.5175, Z -126.0150, A 0, B 90, C 0, E1 0, E2 0, E3 0, E4 0 } C_DIS
LIN{ E6POS: X 704.9347, Y -60.2631, Z -126.0150, A 0, B 90, C 0, E1 0, E2 0, E3 0, E4 0 } C_DIS
LIN{ E6POS: X 704.9603, Y -60.1571, Z -126.0150, A 0, B 90, C 0, E1 0, E2 0, E3 0, E4 0 } C_DIS
LIN{ E6POS: X 705.1554, Y -59.1763, Z -126.0150, A 0, B 90, C 0, E1 0, E2 0, E3 0, E4 0 } C_DIS
LIN{ E6POS: X 705.1971, Y -58.9670, Z -126.0150, A 0, B 90, C 0, E1 0, E2 0, E3 0, E4 0 } C_DIS
LIN{ E6POS: X 705.2218, Y -58.8649, Z -126.0150, A 0, B 90, C 0, E1 0, E2 0, E3 0, E4 0 } C_DIS
LIN{ E6POS: X 705.4108, Y -57.8829, Z -126.0150, A 0, B 90, C 0, E1 0, E2 0, E3 0, E4 0 } C_DIS
LIN{ E6POS: X 705.4510, Y -57.6743, Z -126.0150, A 0, B 90, C 0, E1 0, E2 0, E3 0, E4 0 } C_DIS
LIN{ E6POS: X 705.4749, Y -57.5722, Z -126.0150, A 0, B 90, C 0, E1 0, E2 0, E3 0, E4 0 } C_DIS
LIN{ E6POS: X 705.6553, Y -56.5886, Z -126.0150, A 0, B 90, C 0, E1 0, E2 0, E3 0, E4 0 } C_DIS
LIN{ E6POS: X 705.7008, Y -56.3405, Z -126.0150, A 0, B 90, C 0, E1 0, E2 0, E3 0, E4 0 } C_DIS
LIN{ E6POS: X 705.7241, Y -56.2346, Z -126.0150, A 0, B 90, C 0, E1 0, E2 0, E3 0, E4 0 } C_DIS
LIN{ E6POS: X 705.8940, Y -55.2491, Z -126.0150, A 0, B 90, C 0, E1 0, E2 0, E3 0, E4 0 } C_DIS
LIN{ E6POS: X 705.9512, Y -54.9171, Z -126.0150, A 0, B 90, C 0, E1 0, E2 0, E3 0, E4 0 } C_DIS
LIN{ E6POS: X 705.9741, Y -54.8036, Z -126.0150, A 0, B 90, C 0, E1 0, E2 0, E3 0, E4 0 } C_DIS
LIN{ E6POS: X 706.1373, Y -53.8170, Z -126.0150, A 0, B 90, C 0, E1 0, E2 0, E3 0, E4 0 } C_DIS
LIN{ E6POS: X 706.1990, Y -53.4443, Z -126.0150, A 0, B 90, C 0, E1 0, E2 0, E3 0, E4 0 } C_DIS
LIN{ E6POS: X 706.2213, Y -53.3269, Z -126.0150, A 0, B 90, C 0, E1 0, E2 0, E3 0, E4 0 } C_DIS
LIN{ E6POS: X 706.3796, Y -52.3395, Z -126.0150, A 0, B 90, C 0, E1 0, E2 0, E3 0, E4 0 } C_DIS
LIN{ E6POS: X 706.4391, Y -51.9682, Z -126.0150, A 0, B 90, C 0, E1 0, E2 0, E3 0, E4 0 } C_DIS
LIN{ E6POS: X 706.4608, Y -51.8508, Z -126.0150, A 0, B 90, C 0, E1 0, E2 0, E3 0, E4 0 } C_DIS
LIN{ E6POS: X 706.6168, Y -50.8630, Z -126.0150, A 0, B 90, C 0, E1 0, E2 0, E3 0, E4 0 } C_DIS
LIN{ E6POS: X 706.6687, Y -50.5340, Z -126.0150, A 0, B 90, C 0, E1 0, E2 0, E3 0, E4 0 } C_DIS
LIN{ E6POS: X 706.6899, Y -50.4205, Z -126.0150, A 0, B 90, C 0, E1 0, E2 0, E3 0, E4 0 } C_DIS
LIN{ E6POS: X 706.8452, Y -49.4327, Z -126.0150, A 0, B 90, C 0, E1 0, E2 0, E3 0, E4 0 } C_DIS
LIN{ E6POS: X 706.8833, Y -49.1901, Z -126.0150, A 0, B 90, C 0, E1 0, E2 0, E3 0, E4 0 } C_DIS
LIN{ E6POS: X 706.9038, Y -49.0843, Z -126.0150, A 0, B 90, C 0, E1 0, E2 0, E3 0, E4 0 } C_DIS
LIN{ E6POS: X 707.0597, Y -48.0965, Z -126.0150, A 0, B 90, C 0, E1 0, E2 0, E3 0, E4 0 } C_DIS
LIN{ E6POS: X 707.0838, Y -47.9433, Z -126.0150, A 0, B 90, C 0, E1 0, E2 0, E3 0, E4 0 } C_DIS
LIN{ E6POS: X 707.1037, Y -47.8445, Z -126.0150, A 0, B 90, C 0, E1 0, E2 0, E3 0, E4 0 } C_DIS
LIN{ E6POS: X 707.2617, Y -46.8571, Z -126.0150, A 0, B 90, C 0, E1 0, E2 0, E3 0, E4 0 } C_DIS
LIN{ E6POS: X 707.2707, Y -46.8009, Z -126.0150, A 0, B 90, C 0, E1 0, E2 0, E3 0, E4 0 } C_DIS
LIN{ E6POS: X 707.2898, Y -46.7083, Z -126.0150, A 0, B 90, C 0, E1 0, E2 0, E3 0, E4 0 } C_DIS
LIN{ E6POS: X 707.4573, Y -45.7224, Z -126.0150, A 0, B 90, C 0, E1 0, E2 0, E3 0, E4 0 } C_DIS
LIN{ E6POS: X 707.6248, Y -44.7366, Z -126.0150, A 0, B 90, C 0, E1 0, E2 0, E3 0, E4 0 } C_DIS
LIN{ E6POS: X 707.6588, Y -44.5363, Z -126.0150, A 0, B 90, C 0, E1 0, E2 0, E3 0, E4 0 } C_DIS
LIN{ E6POS: X 707.6770, Y -44.4492, Z -126.0150, A 0, B 90, C 0, E1 0, E2 0, E3 0, E4 0 } C_DIS
LIN{ E6POS: X 707.6943, Y -44.3667, Z -126.0150, A 0, B 90, C 0, E1 0, E2 0, E3 0, E4 0 } C_DIS
LIN{ E6POS: X 707.7109, Y -44.2851, Z -126.0150, A 0, B 90, C 0, E1 0, E2 0, E3 0, E4 0 } C_DIS
LIN{ E6POS: X 707.7271, Y -44.2005, Z -126.0150, A 0, B 90, C 0, E1 0, E2 0, E3 0, E4 0 } C_DIS
LIN{ E6POS: X 707.8900, Y -43.2139, Z -126.0150, A 0, B 90, C 0, E1 0, E2 0, E3 0, E4 0 } C_DIS
LIN{ E6POS: X 708.0530, Y -42.2273, Z -126.0150, A 0, B 90, C 0, E1 0, E2 0, E3 0, E4 0 } C_DIS
LIN{ E6POS: X 708.0783, Y -42.0737, Z -126.0150, A 0, B 90, C 0, E1 0, E2 0, E3 0, E4 0 } C_DIS
LIN{ E6POS: X 708.0945, Y -41.9822, Z -126.0150, A 0, B 90, C 0, E1 0, E2 0, E3 0, E4 0 } C_DIS
LIN{ E6POS: X 708.2337, Y -40.9919, Z -126.0150, A 0, B 90, C 0, E1 0, E2 0, E3 0, E4 0 } C_DIS
LIN{ E6POS: X 708.2437, Y -40.9205, Z -126.0150, A 0, B 90, C 0, E1 0, E2 0, E3 0, E4 0 } C_DIS
LIN{ E6POS: X 708.2599, Y -40.8183, Z -126.0150, A 0, B 90, C 0, E1 0, E2 0, E3 0, E4 0 } C_DIS
LIN{ E6POS: X 708.3881, Y -39.8266, Z -126.0150, A 0, B 90, C 0, E1 0, E2 0, E3 0, E4 0 } C_DIS
LIN{ E6POS: X 708.4105, Y -39.6538, Z -126.0150, A 0, B 90, C 0, E1 0, E2 0, E3 0, E4 0 } C_DIS
LIN{ E6POS: X 708.4267, Y -39.5452, Z -126.0150, A 0, B 90, C 0, E1 0, E2 0, E3 0, E4 0 } C_DIS
LIN{ E6POS: X 708.5478, Y -38.5525, Z -126.0150, A 0, B 90, C 0, E1 0, E2 0, E3 0, E4 0 } C_DIS
LIN{ E6POS: X 708.5753, Y -38.3274, Z -126.0150, A 0, B 90, C 0, E1 0, E2 0, E3 0, E4 0 } C_DIS
LIN{ E6POS: X 708.5911, Y -38.2165, Z -126.0150, A 0, B 90, C 0, E1 0, E2 0, E3 0, E4 0 } C_DIS
LIN{ E6POS: X 708.7062, Y -37.2231, Z -126.0150, A 0, B 90, C 0, E1 0, E2 0, E3 0, E4 0 } C_DIS
LIN{ E6POS: X 708.7323, Y -36.9973, Z -126.0150, A 0, B 90, C 0, E1 0, E2 0, E3 0, E4 0 } C_DIS
LIN{ E6POS: X 708.7476, Y -36.8884, Z -126.0150, A 0, B 90, C 0, E1 0, E2 0, E3 0, E4 0 } C_DIS
LIN{ E6POS: X 708.8563, Y -35.8943, Z -126.0150, A 0, B 90, C 0, E1 0, E2 0, E3 0, E4 0 } C_DIS
LIN{ E6POS: X 708.8757, Y -35.7168, Z -126.0150, A 0, B 90, C 0, E1 0, E2 0, E3 0, E4 0 } C_DIS
LIN{ E6POS: X 708.8902, Y -35.6139, Z -126.0150, A 0, B 90, C 0, E1 0, E2 0, E3 0, E4 0 } C_DIS
LIN{ E6POS: X 708.9930, Y -34.6192, Z -126.0150, A 0, B 90, C 0, E1 0, E2 0, E3 0, E4 0 } C_DIS
LIN{ E6POS: X 709.0095, Y -34.4597, Z -126.0150, A 0, B 90, C 0, E1 0, E2 0, E3 0, E4 0 } C_DIS
LIN{ E6POS: X 709.0235, Y -34.3596, Z -126.0150, A 0, B 90, C 0, E1 0, E2 0, E3 0, E4 0 } C_DIS
LIN{ E6POS: X 709.1221, Y -33.3645, Z -126.0150, A 0, B 90, C 0, E1 0, E2 0, E3 0, E4 0 } C_DIS
LIN{ E6POS: X 709.1397, Y -33.1872, Z -126.0150, A 0, B 90, C 0, E1 0, E2 0, E3 0, E4 0 } C_DIS
LIN{ E6POS: X 709.1532, Y -33.0863, Z -126.0150, A 0, B 90, C 0, E1 0, E2 0, E3 0, E4 0 } C_DIS
LIN{ E6POS: X 709.2469, Y -32.0908, Z -126.0150, A 0, B 90, C 0, E1 0, E2 0, E3 0, E4 0 } C_DIS
LIN{ E6POS: X 709.2683, Y -31.8639, Z -126.0150, A 0, B 90, C 0, E1 0, E2 0, E3 0, E4 0 } C_DIS
LIN{ E6POS: X 709.2815, Y -31.7590, Z -126.0150, A 0, B 90, C 0, E1 0, E2 0, E3 0, E4 0 } C_DIS
LIN{ E6POS: X 709.3725, Y -30.7631, Z -126.0150, A 0, B 90, C 0, E1 0, E2 0, E3 0, E4 0 } C_DIS
LIN{ E6POS: X 709.4009, Y -30.4527, Z -126.0150, A 0, B 90, C 0, E1 0, E2 0, E3 0, E4 0 } C_DIS
LIN{ E6POS: X 709.4139, Y -30.3402, Z -126.0150, A 0, B 90, C 0, E1 0, E2 0, E3 0, E4 0 } C_DIS
LIN{ E6POS: X 709.5023, Y -29.3441, Z -126.0150, A 0, B 90, C 0, E1 0, E2 0, E3 0, E4 0 } C_DIS
LIN{ E6POS: X 709.5335, Y -28.9928, Z -126.0150, A 0, B 90, C 0, E1 0, E2 0, E3 0, E4 0 } C_DIS
LIN{ E6POS: X 709.5464, Y -28.8766, Z -126.0150, A 0, B 90, C 0, E1 0, E2 0, E3 0, E4 0 } C_DIS
LIN{ E6POS: X 709.6322, Y -27.8803, Z -126.0150, A 0, B 90, C 0, E1 0, E2 0, E3 0, E4 0 } C_DIS
LIN{ E6POS: X 709.6623, Y -27.5301, Z -126.0150, A 0, B 90, C 0, E1 0, E2 0, E3 0, E4 0 } C_DIS
LIN{ E6POS: X 709.6748, Y -27.4139, Z -126.0150, A 0, B 90, C 0, E1 0, E2 0, E3 0, E4 0 } C_DIS
LIN{ E6POS: X 709.7570, Y -26.4173, Z -126.0150, A 0, B 90, C 0, E1 0, E2 0, E3 0, E4 0 } C_DIS
LIN{ E6POS: X 709.7824, Y -26.1097, Z -126.0150, A 0, B 90, C 0, E1 0, E2 0, E3 0, E4 0 } C_DIS
LIN{ E6POS: X 709.7945, Y -25.9974, Z -126.0150, A 0, B 90, C 0, E1 0, E2 0, E3 0, E4 0 } C_DIS
LIN{ E6POS: X 709.8731, Y -25.0005, Z -126.0150, A 0, B 90, C 0, E1 0, E2 0, E3 0, E4 0 } C_DIS
LIN{ E6POS: X 709.8906, Y -24.7785, Z -126.0150, A 0, B 90, C 0, E1 0, E2 0, E3 0, E4 0 } C_DIS
LIN{ E6POS: X 709.9021, Y -24.6738, Z -126.0150, A 0, B 90, C 0, E1 0, E2 0, E3 0, E4 0 } C_DIS
LIN{ E6POS: X 709.9763, Y -23.6766, Z -126.0150, A 0, B 90, C 0, E1 0, E2 0, E3 0, E4 0 } C_DIS
LIN{ E6POS: X 709.9888, Y -23.5084, Z -126.0150, A 0, B 90, C 0, E1 0, E2 0, E3 0, E4 0 } C_DIS
LIN{ E6POS: X 709.9997, Y -23.4089, Z -126.0150, A 0, B 90, C 0, E1 0, E2 0, E3 0, E4 0 } C_DIS
LIN{ E6POS: X 710.0694, Y -22.4113, Z -126.0150, A 0, B 90, C 0, E1 0, E2 0, E3 0, E4 0 } C_DIS
LIN{ E6POS: X 710.0798, Y -22.2624, Z -126.0150, A 0, B 90, C 0, E1 0, E2 0, E3 0, E4 0 } C_DIS
LIN{ E6POS: X 710.0901, Y -22.1655, Z -126.0150, A 0, B 90, C 0, E1 0, E2 0, E3 0, E4 0 } C_DIS
LIN{ E6POS: X 710.1562, Y -21.1677, Z -126.0150, A 0, B 90, C 0, E1 0, E2 0, E3 0, E4 0 } C_DIS
LIN{ E6POS: X 710.1667, Y -21.0084, Z -126.0150, A 0, B 90, C 0, E1 0, E2 0, E3 0, E4 0 } C_DIS
LIN{ E6POS: X 710.1764, Y -20.9117, Z -126.0150, A 0, B 90, C 0, E1 0, E2 0, E3 0, E4 0 } C_DIS
LIN{ E6POS: X 710.2396, Y -19.9137, Z -126.0150, A 0, B 90, C 0, E1 0, E2 0, E3 0, E4 0 } C_DIS
LIN{ E6POS: X 710.2526, Y -19.7095, Z -126.0150, A 0, B 90, C 0, E1 0, E2 0, E3 0, E4 0 } C_DIS
LIN{ E6POS: X 710.2615, Y -19.6103, Z -126.0150, A 0, B 90, C 0, E1 0, E2 0, E3 0, E4 0 } C_DIS
LIN{ E6POS: X 710.3221, Y -18.6121, Z -126.0150, A 0, B 90, C 0, E1 0, E2 0, E3 0, E4 0 } C_DIS
LIN{ E6POS: X 710.3365, Y -18.3753, Z -126.0150, A 0, B 90, C 0, E1 0, E2 0, E3 0, E4 0 } C_DIS
LIN{ E6POS: X 710.3449, Y -18.2743, Z -126.0150, A 0, B 90, C 0, E1 0, E2 0, E3 0, E4 0 } C_DIS
LIN{ E6POS: X 710.4050, Y -17.2761, Z -126.0150, A 0, B 90, C 0, E1 0, E2 0, E3 0, E4 0 } C_DIS
LIN{ E6POS: X 710.4206, Y -17.0165, Z -126.0150, A 0, B 90, C 0, E1 0, E2 0, E3 0, E4 0 } C_DIS
LIN{ E6POS: X 710.4286, Y -16.9143, Z -126.0150, A 0, B 90, C 0, E1 0, E2 0, E3 0, E4 0 } C_DIS
LIN{ E6POS: X 710.4914, Y -15.9162, Z -126.0150, A 0, B 90, C 0, E1 0, E2 0, E3 0, E4 0 } C_DIS
LIN{ E6POS: X 710.5474, Y -15.0273, Z -126.0150, A 0, B 90, C 0, E1 0, E2 0, E3 0, E4 0 } C_DIS
LIN{ E6POS: X 710.5615, Y -14.8590, Z -126.0150, A 0, B 90, C 0, E1 0, E2 0, E3 0, E4 0 } C_DIS
LIN{ E6POS: X 710.6181, Y -13.8606, Z -126.0150, A 0, B 90, C 0, E1 0, E2 0, E3 0, E4 0 } C_DIS
LIN{ E6POS: X 710.6747, Y -12.8622, Z -126.0150, A 0, B 90, C 0, E1 0, E2 0, E3 0, E4 0 } C_DIS
LIN{ E6POS: X 710.6884, Y -12.6207, Z -126.0150, A 0, B 90, C 0, E1 0, E2 0, E3 0, E4 0 } C_DIS
LIN{ E6POS: X 710.7077, Y -12.4148, Z -126.0150, A 0, B 90, C 0, E1 0, E2 0, E3 0, E4 0 } C_DIS
LIN{ E6POS: X 710.7573, Y -11.4161, Z -126.0150, A 0, B 90, C 0, E1 0, E2 0, E3 0, E4 0 } C_DIS
LIN{ E6POS: X 710.7617, Y -11.3291, Z -126.0150, A 0, B 90, C 0, E1 0, E2 0, E3 0, E4 0 } C_DIS
LIN{ E6POS: X 710.7698, Y -11.2357, Z -126.0150, A 0, B 90, C 0, E1 0, E2 0, E3 0, E4 0 } C_DIS
LIN{ E6POS: X 710.8179, Y -10.2368, Z -126.0150, A 0, B 90, C 0, E1 0, E2 0, E3 0, E4 0 } C_DIS
LIN{ E6POS: X 710.8278, Y -10.0297, Z -126.0150, A 0, B 90, C 0, E1 0, E2 0, E3 0, E4 0 } C_DIS
LIN{ E6POS: X 710.8361, Y -9.9263, Z -126.0150, A 0, B 90, C 0, E1 0, E2 0, E3 0, E4 0 } C_DIS
LIN{ E6POS: X 710.8832, Y -8.9274, Z -126.0150, A 0, B 90, C 0, E1 0, E2 0, E3 0, E4 0 } C_DIS
LIN{ E6POS: X 710.8968, Y -8.6389, Z -126.0150, A 0, B 90, C 0, E1 0, E2 0, E3 0, E4 0 } C_DIS
LIN{ E6POS: X 710.9048, Y -8.5282, Z -126.0150, A 0, B 90, C 0, E1 0, E2 0, E3 0, E4 0 } C_DIS
LIN{ E6POS: X 710.9512, Y -7.5292, Z -126.0150, A 0, B 90, C 0, E1 0, E2 0, E3 0, E4 0 } C_DIS
LIN{ E6POS: X 710.9664, Y -7.2009, Z -126.0150, A 0, B 90, C 0, E1 0, E2 0, E3 0, E4 0 } C_DIS
LIN{ E6POS: X 710.9741, Y -7.0866, Z -126.0150, A 0, B 90, C 0, E1 0, E2 0, E3 0, E4 0 } C_DIS
LIN{ E6POS: X 711.0181, Y -6.0876, Z -126.0150, A 0, B 90, C 0, E1 0, E2 0, E3 0, E4 0 } C_DIS
LIN{ E6POS: X 711.0325, Y -5.7613, Z -126.0150, A 0, B 90, C 0, E1 0, E2 0, E3 0, E4 0 } C_DIS
LIN{ E6POS: X 711.0401, Y -5.6470, Z -126.0150, A 0, B 90, C 0, E1 0, E2 0, E3 0, E4 0 } C_DIS
LIN{ E6POS: X 711.0832, Y -4.6480, Z -126.0150, A 0, B 90, C 0, E1 0, E2 0, E3 0, E4 0 } C_DIS
LIN{ E6POS: X 711.0955, Y -4.3638, Z -126.0150, A 0, B 90, C 0, E1 0, E2 0, E3 0, E4 0 } C_DIS
LIN{ E6POS: X 711.1030, Y -4.2533, Z -126.0150, A 0, B 90, C 0, E1 0, E2 0, E3 0, E4 0 } C_DIS
LIN{ E6POS: X 711.1441, Y -3.2542, Z -126.0150, A 0, B 90, C 0, E1 0, E2 0, E3 0, E4 0 } C_DIS
LIN{ E6POS: X 711.1523, Y -3.0542, Z -126.0150, A 0, B 90, C 0, E1 0, E2 0, E3 0, E4 0 } C_DIS
LIN{ E6POS: X 711.1598, Y -2.9513, Z -126.0150, A 0, B 90, C 0, E1 0, E2 0, E3 0, E4 0 } C_DIS
LIN{ E6POS: X 711.1990, Y -1.9521, Z -126.0150, A 0, B 90, C 0, E1 0, E2 0, E3 0, E4 0 } C_DIS
LIN{ E6POS: X 711.2051, Y -1.7949, Z -126.0150, A 0, B 90, C 0, E1 0, E2 0, E3 0, E4 0 } C_DIS
LIN{ E6POS: X 711.2125, Y -1.6957, Z -126.0150, A 0, B 90, C 0, E1 0, E2 0, E3 0, E4 0 } C_DIS
LIN{ E6POS: X 711.2499, Y -0.6964, Z -126.0150, A 0, B 90, C 0, E1 0, E2 0, E3 0, E4 0 } C_DIS
LIN{ E6POS: X 711.2557, Y -0.5405, Z -126.0150, A 0, B 90, C 0, E1 0, E2 0, E3 0, E4 0 } C_DIS
LIN{ E6POS: X 711.2630, Y -0.4415, Z -126.0150, A 0, B 90, C 0, E1 0, E2 0, E3 0, E4 0 } C_DIS
LIN{ E6POS: X 711.2994, Y 0.5578, Z -126.0150, A 0, B 90, C 0, E1 0, E2 0, E3 0, E4 0 } C_DIS
LIN{ E6POS: X 711.3065, Y 0.7518, Z -126.0150, A 0, B 90, C 0, E1 0, E2 0, E3 0, E4 0 } C_DIS
LIN{ E6POS: X 711.3135, Y 0.8543, Z -126.0150, A 0, B 90, C 0, E1 0, E2 0, E3 0, E4 0 } C_DIS
LIN{ E6POS: X 711.3491, Y 1.8536, Z -126.0150, A 0, B 90, C 0, E1 0, E2 0, E3 0, E4 0 } C_DIS
LIN{ E6POS: X 711.3589, Y 2.1292, Z -126.0150, A 0, B 90, C 0, E1 0, E2 0, E3 0, E4 0 } C_DIS
LIN{ E6POS: X 711.3656, Y 2.2387, Z -126.0150, A 0, B 90, C 0, E1 0, E2 0, E3 0, E4 0 } C_DIS
LIN{ E6POS: X 711.4018, Y 3.2381, Z -126.0150, A 0, B 90, C 0, E1 0, E2 0, E3 0, E4 0 } C_DIS
LIN{ E6POS: X 711.4131, Y 3.5522, Z -126.0150, A 0, B 90, C 0, E1 0, E2 0, E3 0, E4 0 } C_DIS
LIN{ E6POS: X 711.4196, Y 3.6653, Z -126.0150, A 0, B 90, C 0, E1 0, E2 0, E3 0, E4 0 } C_DIS
LIN{ E6POS: X 711.4542, Y 4.6647, Z -126.0150, A 0, B 90, C 0, E1 0, E2 0, E3 0, E4 0 } C_DIS
LIN{ E6POS: X 711.4651, Y 4.9775, Z -126.0150, A 0, B 90, C 0, E1 0, E2 0, E3 0, E4 0 } C_DIS
LIN{ E6POS: X 711.4714, Y 5.0904, Z -126.0150, A 0, B 90, C 0, E1 0, E2 0, E3 0, E4 0 } C_DIS
LIN{ E6POS: X 711.5055, Y 6.0898, Z -126.0150, A 0, B 90, C 0, E1 0, E2 0, E3 0, E4 0 } C_DIS
LIN{ E6POS: X 711.5147, Y 6.3603, Z -126.0150, A 0, B 90, C 0, E1 0, E2 0, E3 0, E4 0 } C_DIS
LIN{ E6POS: X 711.5211, Y 6.4695, Z -126.0150, A 0, B 90, C 0, E1 0, E2 0, E3 0, E4 0 } C_DIS
LIN{ E6POS: X 711.5549, Y 7.4689, Z -126.0150, A 0, B 90, C 0, E1 0, E2 0, E3 0, E4 0 } C_DIS
LIN{ E6POS: X 711.5612, Y 7.6562, Z -126.0150, A 0, B 90, C 0, E1 0, E2 0, E3 0, E4 0 } C_DIS
LIN{ E6POS: X 711.5679, Y 7.7581, Z -126.0150, A 0, B 90, C 0, E1 0, E2 0, E3 0, E4 0 } C_DIS
LIN{ E6POS: X 711.6000, Y 8.7576, Z -126.0150, A 0, B 90, C 0, E1 0, E2 0, E3 0, E4 0 } C_DIS
LIN{ E6POS: X 711.6047, Y 8.9019, Z -126.0150, A 0, B 90, C 0, E1 0, E2 0, E3 0, E4 0 } C_DIS
LIN{ E6POS: X 711.6113, Y 9.0001, Z -126.0150, A 0, B 90, C 0, E1 0, E2 0, E3 0, E4 0 } C_DIS
LIN{ E6POS: X 711.6439, Y 9.9995, Z -126.0150, A 0, B 90, C 0, E1 0, E2 0, E3 0, E4 0 } C_DIS
LIN{ E6POS: X 711.6485, Y 10.1418, Z -126.0150, A 0, B 90, C 0, E1 0, E2 0, E3 0, E4 0 } C_DIS
LIN{ E6POS: X 711.6551, Y 10.2398, Z -126.0150, A 0, B 90, C 0, E1 0, E2 0, E3 0, E4 0 } C_DIS
LIN{ E6POS: X 711.6869, Y 11.2393, Z -126.0150, A 0, B 90, C 0, E1 0, E2 0, E3 0, E4 0 } C_DIS
LIN{ E6POS: X 711.6926, Y 11.4196, Z -126.0150, A 0, B 90, C 0, E1 0, E2 0, E3 0, E4 0 } C_DIS
LIN{ E6POS: X 711.6991, Y 11.5210, Z -126.0150, A 0, B 90, C 0, E1 0, E2 0, E3 0, E4 0 } C_DIS
LIN{ E6POS: X 711.7321, Y 12.5204, Z -126.0150, A 0, B 90, C 0, E1 0, E2 0, E3 0, E4 0 } C_DIS
LIN{ E6POS: X 711.7407, Y 12.7809, Z -126.0150, A 0, B 90, C 0, E1 0, E2 0, E3 0, E4 0 } C_DIS
LIN{ E6POS: X 711.7468, Y 12.8891, Z -126.0150, A 0, B 90, C 0, E1 0, E2 0, E3 0, E4 0 } C_DIS
LIN{ E6POS: X 711.7797, Y 13.8886, Z -126.0150, A 0, B 90, C 0, E1 0, E2 0, E3 0, E4 0 } C_DIS
LIN{ E6POS: X 711.7895, Y 14.1869, Z -126.0150, A 0, B 90, C 0, E1 0, E2 0, E3 0, E4 0 } C_DIS
LIN{ E6POS: X 711.7955, Y 14.2986, Z -126.0150, A 0, B 90, C 0, E1 0, E2 0, E3 0, E4 0 } C_DIS
LIN{ E6POS: X 711.8288, Y 15.2980, Z -126.0150, A 0, B 90, C 0, E1 0, E2 0, E3 0, E4 0 } C_DIS
LIN{ E6POS: X 711.8387, Y 15.5952, Z -126.0150, A 0, B 90, C 0, E1 0, E2 0, E3 0, E4 0 } C_DIS
LIN{ E6POS: X 711.8448, Y 15.7067, Z -126.0150, A 0, B 90, C 0, E1 0, E2 0, E3 0, E4 0 } C_DIS
LIN{ E6POS: X 711.8783, Y 16.7062, Z -126.0150, A 0, B 90, C 0, E1 0, E2 0, E3 0, E4 0 } C_DIS
LIN{ E6POS: X 711.8868, Y 16.9617, Z -126.0150, A 0, B 90, C 0, E1 0, E2 0, E3 0, E4 0 } C_DIS
LIN{ E6POS: X 711.8930, Y 17.0696, Z -126.0150, A 0, B 90, C 0, E1 0, E2 0, E3 0, E4 0 } C_DIS
LIN{ E6POS: X 711.9268, Y 18.0691, Z -126.0150, A 0, B 90, C 0, E1 0, E2 0, E3 0, E4 0 } C_DIS
LIN{ E6POS: X 711.9326, Y 18.2412, Z -126.0150, A 0, B 90, C 0, E1 0, E2 0, E3 0, E4 0 } C_DIS
LIN{ E6POS: X 711.9392, Y 18.3419, Z -126.0150, A 0, B 90, C 0, E1 0, E2 0, E3 0, E4 0 } C_DIS
LIN{ E6POS: X 711.9723, Y 19.3414, Z -126.0150, A 0, B 90, C 0, E1 0, E2 0, E3 0, E4 0 } C_DIS
LIN{ E6POS: X 711.9766, Y 19.4711, Z -126.0150, A 0, B 90, C 0, E1 0, E2 0, E3 0, E4 0 } C_DIS
LIN{ E6POS: X 711.9833, Y 19.5682, Z -126.0150, A 0, B 90, C 0, E1 0, E2 0, E3 0, E4 0 } C_DIS
LIN{ E6POS: X 712.0175, Y 20.5676, Z -126.0150, A 0, B 90, C 0, E1 0, E2 0, E3 0, E4 0 } C_DIS
LIN{ E6POS: X 712.0219, Y 20.6951, Z -126.0150, A 0, B 90, C 0, E1 0, E2 0, E3 0, E4 0 } C_DIS
LIN{ E6POS: X 712.0286, Y 20.7919, Z -126.0150, A 0, B 90, C 0, E1 0, E2 0, E3 0, E4 0 } C_DIS
LIN{ E6POS: X 712.0649, Y 21.7913, Z -126.0150, A 0, B 90, C 0, E1 0, E2 0, E3 0, E4 0 } C_DIS
LIN{ E6POS: X 712.0709, Y 21.9569, Z -126.0150, A 0, B 90, C 0, E1 0, E2 0, E3 0, E4 0 } C_DIS
LIN{ E6POS: X 712.0776, Y 22.0569, Z -126.0150, A 0, B 90, C 0, E1 0, E2 0, E3 0, E4 0 } C_DIS
LIN{ E6POS: X 712.1144, Y 23.0563, Z -126.0150, A 0, B 90, C 0, E1 0, E2 0, E3 0, E4 0 } C_DIS
LIN{ E6POS: X 712.1233, Y 23.2993, Z -126.0150, A 0, B 90, C 0, E1 0, E2 0, E3 0, E4 0 } C_DIS
LIN{ E6POS: X 712.1298, Y 23.4061, Z -126.0150, A 0, B 90, C 0, E1 0, E2 0, E3 0, E4 0 } C_DIS
LIN{ E6POS: X 712.1711, Y 24.4052, Z -126.0150, A 0, B 90, C 0, E1 0, E2 0, E3 0, E4 0 } C_DIS
LIN{ E6POS: X 712.1814, Y 24.6542, Z -126.0150, A 0, B 90, C 0, E1 0, E2 0, E3 0, E4 0 } C_DIS
LIN{ E6POS: X 712.1879, Y 24.7629, Z -126.0150, A 0, B 90, C 0, E1 0, E2 0, E3 0, E4 0 } C_DIS
LIN{ E6POS: X 712.2335, Y 25.7618, Z -126.0150, A 0, B 90, C 0, E1 0, E2 0, E3 0, E4 0 } C_DIS
LIN{ E6POS: X 712.2418, Y 25.9424, Z -126.0150, A 0, B 90, C 0, E1 0, E2 0, E3 0, E4 0 } C_DIS
LIN{ E6POS: X 712.2485, Y 26.0480, Z -126.0150, A 0, B 90, C 0, E1 0, E2 0, E3 0, E4 0 } C_DIS
LIN{ E6POS: X 712.3163, Y 27.0457, Z -126.0150, A 0, B 90, C 0, E1 0, E2 0, E3 0, E4 0 } C_DIS
LIN{ E6POS: X 712.3841, Y 28.0434, Z -126.0150, A 0, B 90, C 0, E1 0, E2 0, E3 0, E4 0 } C_DIS
LIN{ E6POS: X 712.4007, Y 28.2869, Z -126.0150, A 0, B 90, C 0, E1 0, E2 0, E3 0, E4 0 } C_DIS
LIN{ E6POS: X 712.4079, Y 28.3848, Z -126.0150, A 0, B 90, C 0, E1 0, E2 0, E3 0, E4 0 } C_DIS
LIN{ E6POS: X 712.4156, Y 28.4698, Z -126.0150, A 0, B 90, C 0, E1 0, E2 0, E3 0, E4 0 } C_DIS
LIN{ E6POS: X 712.4237, Y 28.5499, Z -126.0150, A 0, B 90, C 0, E1 0, E2 0, E3 0, E4 0 } C_DIS
LIN{ E6POS: X 712.4319, Y 28.6325, Z -126.0150, A 0, B 90, C 0, E1 0, E2 0, E3 0, E4 0 } C_DIS
LIN{ E6POS: X 712.5014, Y 29.6301, Z -126.0150, A 0, B 90, C 0, E1 0, E2 0, E3 0, E4 0 } C_DIS
LIN{ E6POS: X 712.5710, Y 30.6277, Z -126.0150, A 0, B 90, C 0, E1 0, E2 0, E3 0, E4 0 } C_DIS
LIN{ E6POS: X 712.5858, Y 30.8413, Z -126.0150, A 0, B 90, C 0, E1 0, E2 0, E3 0, E4 0 } C_DIS
LIN{ E6POS: X 712.5938, Y 30.9342, Z -126.0150, A 0, B 90, C 0, E1 0, E2 0, E3 0, E4 0 } C_DIS
LIN{ E6POS: X 712.6348, Y 31.9334, Z -126.0150, A 0, B 90, C 0, E1 0, E2 0, E3 0, E4 0 } C_DIS
LIN{ E6POS: X 712.6494, Y 32.2891, Z -126.0150, A 0, B 90, C 0, E1 0, E2 0, E3 0, E4 0 } C_DIS
LIN{ E6POS: X 712.6568, Y 32.4001, Z -126.0150, A 0, B 90, C 0, E1 0, E2 0, E3 0, E4 0 } C_DIS
LIN{ E6POS: X 712.6924, Y 33.3994, Z -126.0150, A 0, B 90, C 0, E1 0, E2 0, E3 0, E4 0 } C_DIS
LIN{ E6POS: X 712.7111, Y 33.9247, Z -126.0150, A 0, B 90, C 0, E1 0, E2 0, E3 0, E4 0 } C_DIS
LIN{ E6POS: X 712.7183, Y 34.0445, Z -126.0150, A 0, B 90, C 0, E1 0, E2 0, E3 0, E4 0 } C_DIS
LIN{ E6POS: X 712.7543, Y 35.0438, Z -126.0150, A 0, B 90, C 0, E1 0, E2 0, E3 0, E4 0 } C_DIS
LIN{ E6POS: X 712.7731, Y 35.5680, Z -126.0150, A 0, B 90, C 0, E1 0, E2 0, E3 0, E4 0 } C_DIS
LIN{ E6POS: X 712.7805, Y 35.6877, Z -126.0150, A 0, B 90, C 0, E1 0, E2 0, E3 0, E4 0 } C_DIS
LIN{ E6POS: X 712.8238, Y 36.6867, Z -126.0150, A 0, B 90, C 0, E1 0, E2 0, E3 0, E4 0 } C_DIS
LIN{ E6POS: X 712.8391, Y 37.0407, Z -126.0150, A 0, B 90, C 0, E1 0, E2 0, E3 0, E4 0 } C_DIS
LIN{ E6POS: X 712.8469, Y 37.1513, Z -126.0150, A 0, B 90, C 0, E1 0, E2 0, E3 0, E4 0 } C_DIS
LIN{ E6POS: X 712.9212, Y 38.1485, Z -126.0150, A 0, B 90, C 0, E1 0, E2 0, E3 0, E4 0 } C_DIS
LIN{ E6POS: X 712.9847, Y 39.0007, Z -126.0150, A 0, B 90, C 0, E1 0, E2 0, E3 0, E4 0 } C_DIS
LIN{ E6POS: X 712.9933, Y 39.0932, Z -126.0150, A 0, B 90, C 0, E1 0, E2 0, E3 0, E4 0 } C_DIS
LIN{ E6POS: X 713.0024, Y 39.1764, Z -126.0150, A 0, B 90, C 0, E1 0, E2 0, E3 0, E4 0 } C_DIS
LIN{ E6POS: X 713.0119, Y 39.2593, Z -126.0150, A 0, B 90, C 0, E1 0, E2 0, E3 0, E4 0 } C_DIS
LIN{ E6POS: X 713.0950, Y 40.2558, Z -126.0150, A 0, B 90, C 0, E1 0, E2 0, E3 0, E4 0 } C_DIS
LIN{ E6POS: X 713.1650, Y 41.0943, Z -126.0150, A 0, B 90, C 0, E1 0, E2 0, E3 0, E4 0 } C_DIS
LIN{ E6POS: X 713.1747, Y 41.1858, Z -126.0150, A 0, B 90, C 0, E1 0, E2 0, E3 0, E4 0 } C_DIS
LIN{ E6POS: X 713.2371, Y 42.1838, Z -126.0150, A 0, B 90, C 0, E1 0, E2 0, E3 0, E4 0 } C_DIS
LIN{ E6POS: X 713.2580, Y 42.5168, Z -126.0150, A 0, B 90, C 0, E1 0, E2 0, E3 0, E4 0 } C_DIS
LIN{ E6POS: X 713.2674, Y 42.6257, Z -126.0150, A 0, B 90, C 0, E1 0, E2 0, E3 0, E4 0 } C_DIS
LIN{ E6POS: X 713.3234, Y 43.6242, Z -126.0150, A 0, B 90, C 0, E1 0, E2 0, E3 0, E4 0 } C_DIS
LIN{ E6POS: X 713.3532, Y 44.1549, Z -126.0150, A 0, B 90, C 0, E1 0, E2 0, E3 0, E4 0 } C_DIS
LIN{ E6POS: X 713.3628, Y 44.2738, Z -126.0150, A 0, B 90, C 0, E1 0, E2 0, E3 0, E4 0 } C_DIS
LIN{ E6POS: X 713.4172, Y 45.2724, Z -126.0150, A 0, B 90, C 0, E1 0, E2 0, E3 0, E4 0 } C_DIS
LIN{ E6POS: X 713.4494, Y 45.8639, Z -126.0150, A 0, B 90, C 0, E1 0, E2 0, E3 0, E4 0 } C_DIS
LIN{ E6POS: X 713.4592, Y 45.9855, Z -126.0150, A 0, B 90, C 0, E1 0, E2 0, E3 0, E4 0 } C_DIS
LIN{ E6POS: X 713.5160, Y 46.9839, Z -126.0150, A 0, B 90, C 0, E1 0, E2 0, E3 0, E4 0 } C_DIS
LIN{ E6POS: X 713.5456, Y 47.5039, Z -126.0150, A 0, B 90, C 0, E1 0, E2 0, E3 0, E4 0 } C_DIS
LIN{ E6POS: X 713.5555, Y 47.6208, Z -126.0150, A 0, B 90, C 0, E1 0, E2 0, E3 0, E4 0 } C_DIS
LIN{ E6POS: X 713.6207, Y 48.6187, Z -126.0150, A 0, B 90, C 0, E1 0, E2 0, E3 0, E4 0 } C_DIS
LIN{ E6POS: X 713.6410, Y 48.9300, Z -126.0150, A 0, B 90, C 0, E1 0, E2 0, E3 0, E4 0 } C_DIS
LIN{ E6POS: X 713.6513, Y 49.0348, Z -126.0150, A 0, B 90, C 0, E1 0, E2 0, E3 0, E4 0 } C_DIS
LIN{ E6POS: X 713.7250, Y 50.0320, Z -126.0150, A 0, B 90, C 0, E1 0, E2 0, E3 0, E4 0 } C_DIS
LIN{ E6POS: X 713.7366, Y 50.1882, Z -126.0150, A 0, B 90, C 0, E1 0, E2 0, E3 0, E4 0 } C_DIS
LIN{ E6POS: X 713.7470, Y 50.2837, Z -126.0150, A 0, B 90, C 0, E1 0, E2 0, E3 0, E4 0 } C_DIS
LIN{ E6POS: X 713.8273, Y 51.2805, Z -126.0150, A 0, B 90, C 0, E1 0, E2 0, E3 0, E4 0 } C_DIS
LIN{ E6POS: X 713.8316, Y 51.3331, Z -126.0150, A 0, B 90, C 0, E1 0, E2 0, E3 0, E4 0 } C_DIS
LIN{ E6POS: X 713.8423, Y 51.4226, Z -126.0150, A 0, B 90, C 0, E1 0, E2 0, E3 0, E4 0 } C_DIS
LIN{ E6POS: X 713.9264, Y 52.4190, Z -126.0150, A 0, B 90, C 0, E1 0, E2 0, E3 0, E4 0 } C_DIS
LIN{ E6POS: X 713.9274, Y 52.4307, Z -126.0150, A 0, B 90, C 0, E1 0, E2 0, E3 0, E4 0 } C_DIS
LIN{ E6POS: X 713.9559, Y 52.5149, Z -126.0150, A 0, B 90, C 0, E1 0, E2 0, E3 0, E4 0 } C_DIS
LIN{ E6POS: X 714.8413, Y 52.3217, Z -126.0150, A 0, B 90, C 0, E1 0, E2 0, E3 0, E4 0 } C_DIS
LIN{ E6POS: X 715.8072, Y 52.0628, Z -126.0150, A 0, B 90, C 0, E1 0, E2 0, E3 0, E4 0 } C_DIS
LIN{ E6POS: X 716.7731, Y 51.8039, Z -126.0150, A 0, B 90, C 0, E1 0, E2 0, E3 0, E4 0 } C_DIS
LIN{ E6POS: X 717.4810, Y 51.6142, Z -126.0150, A 0, B 90, C 0, E1 0, E2 0, E3 0, E4 0 } C_DIS
LIN{ E6POS: X 717.7422, Y 51.5451, Z -126.0150, A 0, B 90, C 0, E1 0, E2 0, E3 0, E4 0 } C_DIS
LIN{ E6POS: X 718.7066, Y 51.2805, Z -126.0150, A 0, B 90, C 0, E1 0, E2 0, E3 0, E4 0 } C_DIS
LIN{ E6POS: X 719.6710, Y 51.0160, Z -126.0150, A 0, B 90, C 0, E1 0, E2 0, E3 0, E4 0 } C_DIS
LIN{ E6POS: X 720.6354, Y 50.7514, Z -126.0150, A 0, B 90, C 0, E1 0, E2 0, E3 0, E4 0 } C_DIS
LIN{ E6POS: X 721.5997, Y 50.4869, Z -126.0150, A 0, B 90, C 0, E1 0, E2 0, E3 0, E4 0 } C_DIS
LIN{ E6POS: X 722.5641, Y 50.2224, Z -126.0150, A 0, B 90, C 0, E1 0, E2 0, E3 0, E4 0 } C_DIS
LIN{ E6POS: X 723.0176, Y 50.0980, Z -126.0150, A 0, B 90, C 0, E1 0, E2 0, E3 0, E4 0 } C_DIS
LIN{ E6POS: X 723.4344, Y 49.9765, Z -126.0150, A 0, B 90, C 0, E1 0, E2 0, E3 0, E4 0 } C_DIS
LIN{ E6POS: X 724.3982, Y 49.7099, Z -126.0150, A 0, B 90, C 0, E1 0, E2 0, E3 0, E4 0 } C_DIS
LIN{ E6POS: X 725.3620, Y 49.4433, Z -126.0150, A 0, B 90, C 0, E1 0, E2 0, E3 0, E4 0 } C_DIS
LIN{ E6POS: X 726.3258, Y 49.1767, Z -126.0150, A 0, B 90, C 0, E1 0, E2 0, E3 0, E4 0 } C_DIS
LIN{ E6POS: X 727.2896, Y 48.9101, Z -126.0150, A 0, B 90, C 0, E1 0, E2 0, E3 0, E4 0 } C_DIS
LIN{ E6POS: X 728.2534, Y 48.6434, Z -126.0150, A 0, B 90, C 0, E1 0, E2 0, E3 0, E4 0 } C_DIS
LIN{ E6POS: X 729.2172, Y 48.3768, Z -126.0150, A 0, B 90, C 0, E1 0, E2 0, E3 0, E4 0 } C_DIS
LIN{ E6POS: X 730.1810, Y 48.1102, Z -126.0150, A 0, B 90, C 0, E1 0, E2 0, E3 0, E4 0 } C_DIS
LIN{ E6POS: X 731.1448, Y 47.8436, Z -126.0150, A 0, B 90, C 0, E1 0, E2 0, E3 0, E4 0 } C_DIS
LIN{ E6POS: X 732.1086, Y 47.5770, Z -126.0150, A 0, B 90, C 0, E1 0, E2 0, E3 0, E4 0 } C_DIS
LIN{ E6POS: X 732.2253, Y 47.5447, Z -126.0150, A 0, B 90, C 0, E1 0, E2 0, E3 0, E4 0 } C_DIS
LIN{ E6POS: X 732.9195, Y 47.3396, Z -126.0150, A 0, B 90, C 0, E1 0, E2 0, E3 0, E4 0 } C_DIS
LIN{ E6POS: X 733.8862, Y 47.0838, Z -126.0150, A 0, B 90, C 0, E1 0, E2 0, E3 0, E4 0 } C_DIS
LIN{ E6POS: X 734.8530, Y 46.8281, Z -126.0150, A 0, B 90, C 0, E1 0, E2 0, E3 0, E4 0 } C_DIS
LIN{ E6POS: X 735.8197, Y 46.5723, Z -126.0150, A 0, B 90, C 0, E1 0, E2 0, E3 0, E4 0 } C_DIS
LIN{ E6POS: X 736.7865, Y 46.3165, Z -126.0150, A 0, B 90, C 0, E1 0, E2 0, E3 0, E4 0 } C_DIS
LIN{ E6POS: X 737.7532, Y 46.0608, Z -126.0150, A 0, B 90, C 0, E1 0, E2 0, E3 0, E4 0 } C_DIS
LIN{ E6POS: X 738.7199, Y 45.8050, Z -126.0150, A 0, B 90, C 0, E1 0, E2 0, E3 0, E4 0 } C_DIS
LIN{ E6POS: X 739.6867, Y 45.5492, Z -126.0150, A 0, B 90, C 0, E1 0, E2 0, E3 0, E4 0 } C_DIS
LIN{ E6POS: X 740.6534, Y 45.2934, Z -126.0150, A 0, B 90, C 0, E1 0, E2 0, E3 0, E4 0 } C_DIS
LIN{ E6POS: X 741.6201, Y 45.0377, Z -126.0150, A 0, B 90, C 0, E1 0, E2 0, E3 0, E4 0 } C_DIS
LIN{ E6POS: X 742.5869, Y 44.7819, Z -126.0150, A 0, B 90, C 0, E1 0, E2 0, E3 0, E4 0 } C_DIS
LIN{ E6POS: X 743.5536, Y 44.5261, Z -126.0150, A 0, B 90, C 0, E1 0, E2 0, E3 0, E4 0 } C_DIS
LIN{ E6POS: X 743.8131, Y 44.4575, Z -126.0150, A 0, B 90, C 0, E1 0, E2 0, E3 0, E4 0 } C_DIS
LIN{ E6POS: X 744.6763, Y 44.2142, Z -126.0150, A 0, B 90, C 0, E1 0, E2 0, E3 0, E4 0 } C_DIS
LIN{ E6POS: X 745.6484, Y 43.9798, Z -126.0150, A 0, B 90, C 0, E1 0, E2 0, E3 0, E4 0 } C_DIS
LIN{ E6POS: X 746.6206, Y 43.7454, Z -126.0150, A 0, B 90, C 0, E1 0, E2 0, E3 0, E4 0 } C_DIS
LIN{ E6POS: X 747.5927, Y 43.5109, Z -126.0150, A 0, B 90, C 0, E1 0, E2 0, E3 0, E4 0 } C_DIS
LIN{ E6POS: X 748.5648, Y 43.2765, Z -126.0150, A 0, B 90, C 0, E1 0, E2 0, E3 0, E4 0 } C_DIS
LIN{ E6POS: X 749.5369, Y 43.0420, Z -126.0150, A 0, B 90, C 0, E1 0, E2 0, E3 0, E4 0 } C_DIS
LIN{ E6POS: X 750.5091, Y 42.8076, Z -126.0150, A 0, B 90, C 0, E1 0, E2 0, E3 0, E4 0 } C_DIS
LIN{ E6POS: X 751.4812, Y 42.5731, Z -126.0150, A 0, B 90, C 0, E1 0, E2 0, E3 0, E4 0 } C_DIS
LIN{ E6POS: X 752.4533, Y 42.3387, Z -126.0150, A 0, B 90, C 0, E1 0, E2 0, E3 0, E4 0 } C_DIS
LIN{ E6POS: X 753.4255, Y 42.1042, Z -126.0150, A 0, B 90, C 0, E1 0, E2 0, E3 0, E4 0 } C_DIS
LIN{ E6POS: X 754.3976, Y 41.8698, Z -126.0150, A 0, B 90, C 0, E1 0, E2 0, E3 0, E4 0 } C_DIS
LIN{ E6POS: X 755.3697, Y 41.6353, Z -126.0150, A 0, B 90, C 0, E1 0, E2 0, E3 0, E4 0 } C_DIS
LIN{ E6POS: X 756.2657, Y 41.4192, Z -126.0150, A 0, B 90, C 0, E1 0, E2 0, E3 0, E4 0 } C_DIS
LIN{ E6POS: X 757.1891, Y 41.1833, Z -126.0150, A 0, B 90, C 0, E1 0, E2 0, E3 0, E4 0 } C_DIS
LIN{ E6POS: X 758.1697, Y 40.9873, Z -126.0150, A 0, B 90, C 0, E1 0, E2 0, E3 0, E4 0 } C_DIS
LIN{ E6POS: X 759.1503, Y 40.7912, Z -126.0150, A 0, B 90, C 0, E1 0, E2 0, E3 0, E4 0 } C_DIS
LIN{ E6POS: X 760.1309, Y 40.5952, Z -126.0150, A 0, B 90, C 0, E1 0, E2 0, E3 0, E4 0 } C_DIS
LIN{ E6POS: X 761.1115, Y 40.3992, Z -126.0150, A 0, B 90, C 0, E1 0, E2 0, E3 0, E4 0 } C_DIS
LIN{ E6POS: X 762.0921, Y 40.2031, Z -126.0150, A 0, B 90, C 0, E1 0, E2 0, E3 0, E4 0 } C_DIS
LIN{ E6POS: X 763.0727, Y 40.0071, Z -126.0150, A 0, B 90, C 0, E1 0, E2 0, E3 0, E4 0 } C_DIS
LIN{ E6POS: X 764.0533, Y 39.8110, Z -126.0150, A 0, B 90, C 0, E1 0, E2 0, E3 0, E4 0 } C_DIS
LIN{ E6POS: X 765.0339, Y 39.6150, Z -126.0150, A 0, B 90, C 0, E1 0, E2 0, E3 0, E4 0 } C_DIS
LIN{ E6POS: X 766.0145, Y 39.4190, Z -126.0150, A 0, B 90, C 0, E1 0, E2 0, E3 0, E4 0 } C_DIS
LIN{ E6POS: X 766.9951, Y 39.2229, Z -126.0150, A 0, B 90, C 0, E1 0, E2 0, E3 0, E4 0 } C_DIS
LIN{ E6POS: X 767.9757, Y 39.0269, Z -126.0150, A 0, B 90, C 0, E1 0, E2 0, E3 0, E4 0 } C_DIS
LIN{ E6POS: X 768.0622, Y 39.0096, Z -126.0150, A 0, B 90, C 0, E1 0, E2 0, E3 0, E4 0 } C_DIS
LIN{ E6POS: X 768.9375, Y 38.8265, Z -126.0150, A 0, B 90, C 0, E1 0, E2 0, E3 0, E4 0 } C_DIS
LIN{ E6POS: X 769.9308, Y 38.7114, Z -126.0150, A 0, B 90, C 0, E1 0, E2 0, E3 0, E4 0 } C_DIS
LIN{ E6POS: X 770.9242, Y 38.5962, Z -126.0150, A 0, B 90, C 0, E1 0, E2 0, E3 0, E4 0 } C_DIS
LIN{ E6POS: X 771.9175, Y 38.4810, Z -126.0150, A 0, B 90, C 0, E1 0, E2 0, E3 0, E4 0 } C_DIS
LIN{ E6POS: X 772.9109, Y 38.3659, Z -126.0150, A 0, B 90, C 0, E1 0, E2 0, E3 0, E4 0 } C_DIS
LIN{ E6POS: X 773.9042, Y 38.2507, Z -126.0150, A 0, B 90, C 0, E1 0, E2 0, E3 0, E4 0 } C_DIS
LIN{ E6POS: X 774.8975, Y 38.1356, Z -126.0150, A 0, B 90, C 0, E1 0, E2 0, E3 0, E4 0 } C_DIS
LIN{ E6POS: X 775.8909, Y 38.0204, Z -126.0150, A 0, B 90, C 0, E1 0, E2 0, E3 0, E4 0 } C_DIS
LIN{ E6POS: X 776.8842, Y 37.9052, Z -126.0150, A 0, B 90, C 0, E1 0, E2 0, E3 0, E4 0 } C_DIS
LIN{ E6POS: X 777.6841, Y 37.8125, Z -126.0150, A 0, B 90, C 0, E1 0, E2 0, E3 0, E4 0 } C_DIS
LIN{ E6POS: X 778.4026, Y 37.7278, Z -126.0150, A 0, B 90, C 0, E1 0, E2 0, E3 0, E4 0 } C_DIS
LIN{ E6POS: X 779.4024, Y 37.7073, Z -126.0150, A 0, B 90, C 0, E1 0, E2 0, E3 0, E4 0 } C_DIS
LIN{ E6POS: X 780.4022, Y 37.6868, Z -126.0150, A 0, B 90, C 0, E1 0, E2 0, E3 0, E4 0 } C_DIS
LIN{ E6POS: X 781.4020, Y 37.6664, Z -126.0150, A 0, B 90, C 0, E1 0, E2 0, E3 0, E4 0 } C_DIS
LIN{ E6POS: X 782.4018, Y 37.6459, Z -126.0150, A 0, B 90, C 0, E1 0, E2 0, E3 0, E4 0 } C_DIS
LIN{ E6POS: X 783.4016, Y 37.6254, Z -126.0150, A 0, B 90, C 0, E1 0, E2 0, E3 0, E4 0 } C_DIS
LIN{ E6POS: X 784.4013, Y 37.6050, Z -126.0150, A 0, B 90, C 0, E1 0, E2 0, E3 0, E4 0 } C_DIS
LIN{ E6POS: X 785.4011, Y 37.5845, Z -126.0150, A 0, B 90, C 0, E1 0, E2 0, E3 0, E4 0 } C_DIS
LIN{ E6POS: X 785.5551, Y 37.5813, Z -126.0150, A 0, B 90, C 0, E1 0, E2 0, E3 0, E4 0 } C_DIS
LIN{ E6POS: X 786.1560, Y 37.5704, Z -126.0150, A 0, B 90, C 0, E1 0, E2 0, E3 0, E4 0 } C_DIS
LIN{ E6POS: X 787.1535, Y 37.6412, Z -126.0150, A 0, B 90, C 0, E1 0, E2 0, E3 0, E4 0 } C_DIS
LIN{ E6POS: X 788.1510, Y 37.7120, Z -126.0150, A 0, B 90, C 0, E1 0, E2 0, E3 0, E4 0 } C_DIS
LIN{ E6POS: X 789.1485, Y 37.7828, Z -126.0150, A 0, B 90, C 0, E1 0, E2 0, E3 0, E4 0 } C_DIS
LIN{ E6POS: X 790.1460, Y 37.8536, Z -126.0150, A 0, B 90, C 0, E1 0, E2 0, E3 0, E4 0 } C_DIS
LIN{ E6POS: X 791.1435, Y 37.9244, Z -126.0150, A 0, B 90, C 0, E1 0, E2 0, E3 0, E4 0 } C_DIS
LIN{ E6POS: X 792.1410, Y 37.9952, Z -126.0150, A 0, B 90, C 0, E1 0, E2 0, E3 0, E4 0 } C_DIS
LIN{ E6POS: X 792.2459, Y 38.0027, Z -126.0150, A 0, B 90, C 0, E1 0, E2 0, E3 0, E4 0 } C_DIS
LIN{ E6POS: X 792.7685, Y 38.0409, Z -126.0150, A 0, B 90, C 0, E1 0, E2 0, E3 0, E4 0 } C_DIS
LIN{ E6POS: X 793.7601, Y 38.1698, Z -126.0150, A 0, B 90, C 0, E1 0, E2 0, E3 0, E4 0 } C_DIS
LIN{ E6POS: X 794.7518, Y 38.2986, Z -126.0150, A 0, B 90, C 0, E1 0, E2 0, E3 0, E4 0 } C_DIS
LIN{ E6POS: X 795.7435, Y 38.4275, Z -126.0150, A 0, B 90, C 0, E1 0, E2 0, E3 0, E4 0 } C_DIS
LIN{ E6POS: X 796.7351, Y 38.5564, Z -126.0150, A 0, B 90, C 0, E1 0, E2 0, E3 0, E4 0 } C_DIS
LIN{ E6POS: X 797.7268, Y 38.6853, Z -126.0150, A 0, B 90, C 0, E1 0, E2 0, E3 0, E4 0 } C_DIS
LIN{ E6POS: X 798.3264, Y 38.7632, Z -126.0150, A 0, B 90, C 0, E1 0, E2 0, E3 0, E4 0 } C_DIS
LIN{ E6POS: X 798.8097, Y 38.8260, Z -126.0150, A 0, B 90, C 0, E1 0, E2 0, E3 0, E4 0 } C_DIS
LIN{ E6POS: X 798.7068, Y 37.8313, Z -126.0150, A 0, B 90, C 0, E1 0, E2 0, E3 0, E4 0 } C_DIS
LIN{ E6POS: X 798.6040, Y 36.8366, Z -126.0150, A 0, B 90, C 0, E1 0, E2 0, E3 0, E4 0 } C_DIS
LIN{ E6POS: X 798.5012, Y 35.8419, Z -126.0150, A 0, B 90, C 0, E1 0, E2 0, E3 0, E4 0 } C_DIS
LIN{ E6POS: X 798.3983, Y 34.8472, Z -126.0150, A 0, B 90, C 0, E1 0, E2 0, E3 0, E4 0 } C_DIS
LIN{ E6POS: X 798.2955, Y 33.8525, Z -126.0150, A 0, B 90, C 0, E1 0, E2 0, E3 0, E4 0 } C_DIS
LIN{ E6POS: X 798.1927, Y 32.8578, Z -126.0150, A 0, B 90, C 0, E1 0, E2 0, E3 0, E4 0 } C_DIS
LIN{ E6POS: X 798.0898, Y 31.8631, Z -126.0150, A 0, B 90, C 0, E1 0, E2 0, E3 0, E4 0 } C_DIS
LIN{ E6POS: X 797.9870, Y 30.8684, Z -126.0150, A 0, B 90, C 0, E1 0, E2 0, E3 0, E4 0 } C_DIS
LIN{ E6POS: X 797.8842, Y 29.8737, Z -126.0150, A 0, B 90, C 0, E1 0, E2 0, E3 0, E4 0 } C_DIS
LIN{ E6POS: X 797.7813, Y 28.8790, Z -126.0150, A 0, B 90, C 0, E1 0, E2 0, E3 0, E4 0 } C_DIS
LIN{ E6POS: X 797.6785, Y 27.8843, Z -126.0150, A 0, B 90, C 0, E1 0, E2 0, E3 0, E4 0 } C_DIS
LIN{ E6POS: X 797.5757, Y 26.8896, Z -126.0150, A 0, B 90, C 0, E1 0, E2 0, E3 0, E4 0 } C_DIS
LIN{ E6POS: X 797.4728, Y 25.8949, Z -126.0150, A 0, B 90, C 0, E1 0, E2 0, E3 0, E4 0 } C_DIS
LIN{ E6POS: X 797.3700, Y 24.9002, Z -126.0150, A 0, B 90, C 0, E1 0, E2 0, E3 0, E4 0 } C_DIS
LIN{ E6POS: X 797.2672, Y 23.9055, Z -126.0150, A 0, B 90, C 0, E1 0, E2 0, E3 0, E4 0 } C_DIS
LIN{ E6POS: X 797.2574, Y 23.8108, Z -126.0150, A 0, B 90, C 0, E1 0, E2 0, E3 0, E4 0 } C_DIS
LIN{ E6POS: X 797.1545, Y 22.8161, Z -126.0150, A 0, B 90, C 0, E1 0, E2 0, E3 0, E4 0 } C_DIS
LIN{ E6POS: X 797.1224, Y 22.5051, Z -126.0150, A 0, B 90, C 0, E1 0, E2 0, E3 0, E4 0 } C_DIS
LIN{ E6POS: X 797.0002, Y 21.5126, Z -126.0150, A 0, B 90, C 0, E1 0, E2 0, E3 0, E4 0 } C_DIS
LIN{ E6POS: X 796.8780, Y 20.5201, Z -126.0150, A 0, B 90, C 0, E1 0, E2 0, E3 0, E4 0 } C_DIS
LIN{ E6POS: X 796.7559, Y 19.5276, Z -126.0150, A 0, B 90, C 0, E1 0, E2 0, E3 0, E4 0 } C_DIS
LIN{ E6POS: X 796.6337, Y 18.5351, Z -126.0150, A 0, B 90, C 0, E1 0, E2 0, E3 0, E4 0 } C_DIS
LIN{ E6POS: X 796.5115, Y 17.5426, Z -126.0150, A 0, B 90, C 0, E1 0, E2 0, E3 0, E4 0 } C_DIS
LIN{ E6POS: X 796.3893, Y 16.5500, Z -126.0150, A 0, B 90, C 0, E1 0, E2 0, E3 0, E4 0 } C_DIS
LIN{ E6POS: X 796.2672, Y 15.5575, Z -126.0150, A 0, B 90, C 0, E1 0, E2 0, E3 0, E4 0 } C_DIS
LIN{ E6POS: X 796.1450, Y 14.5650, Z -126.0150, A 0, B 90, C 0, E1 0, E2 0, E3 0, E4 0 } C_DIS
LIN{ E6POS: X 796.0228, Y 13.5725, Z -126.0150, A 0, B 90, C 0, E1 0, E2 0, E3 0, E4 0 } C_DIS
LIN{ E6POS: X 795.9006, Y 12.5800, Z -126.0150, A 0, B 90, C 0, E1 0, E2 0, E3 0, E4 0 } C_DIS
LIN{ E6POS: X 795.7785, Y 11.5875, Z -126.0150, A 0, B 90, C 0, E1 0, E2 0, E3 0, E4 0 } C_DIS
LIN{ E6POS: X 795.6563, Y 10.5950, Z -126.0150, A 0, B 90, C 0, E1 0, E2 0, E3 0, E4 0 } C_DIS
LIN{ E6POS: X 795.5341, Y 9.6025, Z -126.0150, A 0, B 90, C 0, E1 0, E2 0, E3 0, E4 0 } C_DIS
LIN{ E6POS: X 795.4119, Y 8.6100, Z -126.0150, A 0, B 90, C 0, E1 0, E2 0, E3 0, E4 0 } C_DIS
LIN{ E6POS: X 795.4055, Y 8.5580, Z -126.0150, A 0, B 90, C 0, E1 0, E2 0, E3 0, E4 0 } C_DIS
LIN{ E6POS: X 795.2833, Y 7.5655, Z -126.0150, A 0, B 90, C 0, E1 0, E2 0, E3 0, E4 0 } C_DIS
LIN{ E6POS: X 795.2562, Y 7.3452, Z -124.0150, A 0, B 90, C 0, E1 0, E2 0, E3 0, E4 0 } C_DIS
LIN{ E6POS: X 795.0854, Y 6.3599, Z -124.0150, A 0, B 90, C 0, E1 0, E2 0, E3 0, E4 0 } C_DIS
LIN{ E6POS: X 794.9146, Y 5.3746, Z -124.0150, A 0, B 90, C 0, E1 0, E2 0, E3 0, E4 0 } C_DIS
LIN{ E6POS: X 794.7438, Y 4.3893, Z -124.0150, A 0, B 90, C 0, E1 0, E2 0, E3 0, E4 0 } C_DIS
LIN{ E6POS: X 794.5730, Y 3.4040, Z -124.0150, A 0, B 90, C 0, E1 0, E2 0, E3 0, E4 0 } C_DIS
LIN{ E6POS: X 794.4021, Y 2.4187, Z -124.0150, A 0, B 90, C 0, E1 0, E2 0, E3 0, E4 0 } C_DIS
LIN{ E6POS: X 794.2313, Y 1.4334, Z -124.0150, A 0, B 90, C 0, E1 0, E2 0, E3 0, E4 0 } C_DIS
LIN{ E6POS: X 794.0605, Y 0.4481, Z -124.0150, A 0, B 90, C 0, E1 0, E2 0, E3 0, E4 0 } C_DIS
LIN{ E6POS: X 793.8897, Y -0.5372, Z -124.0150, A 0, B 90, C 0, E1 0, E2 0, E3 0, E4 0 } C_DIS
LIN{ E6POS: X 793.7189, Y -1.5225, Z -124.0150, A 0, B 90, C 0, E1 0, E2 0, E3 0, E4 0 } C_DIS
LIN{ E6POS: X 793.5481, Y -2.5078, Z -124.0150, A 0, B 90, C 0, E1 0, E2 0, E3 0, E4 0 } C_DIS
LIN{ E6POS: X 793.3772, Y -3.4931, Z -124.0150, A 0, B 90, C 0, E1 0, E2 0, E3 0, E4 0 } C_DIS
LIN{ E6POS: X 793.2064, Y -4.4784, Z -124.0150, A 0, B 90, C 0, E1 0, E2 0, E3 0, E4 0 } C_DIS
LIN{ E6POS: X 793.0356, Y -5.4637, Z -124.0150, A 0, B 90, C 0, E1 0, E2 0, E3 0, E4 0 } C_DIS
LIN{ E6POS: X 793.0310, Y -5.4900, Z -124.0150, A 0, B 90, C 0, E1 0, E2 0, E3 0, E4 0 } C_DIS
LIN{ E6POS: X 793.0310, Y -5.4900, Z -124.0150, A 0, B 90, C 0, E1 0, E2 0, E3 0, E4 0 } C_DIS
LIN{ E6POS: X 792.7476, Y -6.4490, Z -124.0150, A 0, B 90, C 0, E1 0, E2 0, E3 0, E4 0 } C_DIS
LIN{ E6POS: X 792.4642, Y -7.4080, Z -124.0150, A 0, B 90, C 0, E1 0, E2 0, E3 0, E4 0 } C_DIS
LIN{ E6POS: X 792.1808, Y -8.3670, Z -124.0150, A 0, B 90, C 0, E1 0, E2 0, E3 0, E4 0 } C_DIS
LIN{ E6POS: X 791.8974, Y -9.3260, Z -124.0150, A 0, B 90, C 0, E1 0, E2 0, E3 0, E4 0 } C_DIS
LIN{ E6POS: X 791.6139, Y -10.2850, Z -124.0150, A 0, B 90, C 0, E1 0, E2 0, E3 0, E4 0 } C_DIS
LIN{ E6POS: X 791.3305, Y -11.2440, Z -124.0150, A 0, B 90, C 0, E1 0, E2 0, E3 0, E4 0 } C_DIS
LIN{ E6POS: X 791.0471, Y -12.2030, Z -124.0150, A 0, B 90, C 0, E1 0, E2 0, E3 0, E4 0 } C_DIS
LIN{ E6POS: X 790.7637, Y -13.1620, Z -124.0150, A 0, B 90, C 0, E1 0, E2 0, E3 0, E4 0 } C_DIS
LIN{ E6POS: X 790.4803, Y -14.1210, Z -124.0150, A 0, B 90, C 0, E1 0, E2 0, E3 0, E4 0 } C_DIS
LIN{ E6POS: X 790.2681, Y -14.8387, Z -124.0150, A 0, B 90, C 0, E1 0, E2 0, E3 0, E4 0 } C_DIS
LIN{ E6POS: X 790.2681, Y -14.8387, Z -124.0150, A 0, B 90, C 0, E1 0, E2 0, E3 0, E4 0 } C_DIS
LIN{ E6POS: X 789.6733, Y -15.6426, Z -124.0150, A 0, B 90, C 0, E1 0, E2 0, E3 0, E4 0 } C_DIS
LIN{ E6POS: X 789.0784, Y -16.4464, Z -124.0150, A 0, B 90, C 0, E1 0, E2 0, E3 0, E4 0 } C_DIS
LIN{ E6POS: X 788.4835, Y -17.2502, Z -124.0150, A 0, B 90, C 0, E1 0, E2 0, E3 0, E4 0 } C_DIS
LIN{ E6POS: X 787.8887, Y -18.0540, Z -124.0150, A 0, B 90, C 0, E1 0, E2 0, E3 0, E4 0 } C_DIS
LIN{ E6POS: X 787.2938, Y -18.8579, Z -124.0150, A 0, B 90, C 0, E1 0, E2 0, E3 0, E4 0 } C_DIS
LIN{ E6POS: X 786.7884, Y -19.5408, Z -124.0150, A 0, B 90, C 0, E1 0, E2 0, E3 0, E4 0 } C_DIS
LIN{ E6POS: X 786.7884, Y -19.5408, Z -124.0150, A 0, B 90, C 0, E1 0, E2 0, E3 0, E4 0 } C_DIS
LIN{ E6POS: X 785.8324, Y -19.8339, Z -124.0150, A 0, B 90, C 0, E1 0, E2 0, E3 0, E4 0 } C_DIS
LIN{ E6POS: X 784.8763, Y -20.1271, Z -124.0150, A 0, B 90, C 0, E1 0, E2 0, E3 0, E4 0 } C_DIS
LIN{ E6POS: X 783.9202, Y -20.4202, Z -124.0150, A 0, B 90, C 0, E1 0, E2 0, E3 0, E4 0 } C_DIS
LIN{ E6POS: X 782.9642, Y -20.7133, Z -124.0150, A 0, B 90, C 0, E1 0, E2 0, E3 0, E4 0 } C_DIS
LIN{ E6POS: X 782.4218, Y -20.8796, Z -124.0150, A 0, B 90, C 0, E1 0, E2 0, E3 0, E4 0 } C_DIS
LIN{ E6POS: X 782.4218, Y -20.8796, Z -124.0150, A 0, B 90, C 0, E1 0, E2 0, E3 0, E4 0 } C_DIS
LIN{ E6POS: X 782.4218, Y -20.8796, Z -124.0150, A 0, B 90, C 0, E1 0, E2 0, E3 0, E4 0 } C_DIS
LIN{ E6POS: X 781.4310, Y -20.7447, Z -124.0150, A 0, B 90, C 0, E1 0, E2 0, E3 0, E4 0 } C_DIS
LIN{ E6POS: X 780.4401, Y -20.6098, Z -124.0150, A 0, B 90, C 0, E1 0, E2 0, E3 0, E4 0 } C_DIS
LIN{ E6POS: X 779.4493, Y -20.4749, Z -124.0150, A 0, B 90, C 0, E1 0, E2 0, E3 0, E4 0 } C_DIS
LIN{ E6POS: X 778.4584, Y -20.3400, Z -124.0150, A 0, B 90, C 0, E1 0, E2 0, E3 0, E4 0 } C_DIS
LIN{ E6POS: X 777.4675, Y -20.2051, Z -124.0150, A 0, B 90, C 0, E1 0, E2 0, E3 0, E4 0 } C_DIS
LIN{ E6POS: X 776.9995, Y -20.1414, Z -124.0150, A 0, B 90, C 0, E1 0, E2 0, E3 0, E4 0 } C_DIS
LIN{ E6POS: X 776.9995, Y -20.1414, Z -124.0150, A 0, B 90, C 0, E1 0, E2 0, E3 0, E4 0 } C_DIS
LIN{ E6POS: X 776.0250, Y -19.9173, Z -124.0150, A 0, B 90, C 0, E1 0, E2 0, E3 0, E4 0 } C_DIS
LIN{ E6POS: X 775.0504, Y -19.6932, Z -124.0150, A 0, B 90, C 0, E1 0, E2 0, E3 0, E4 0 } C_DIS
LIN{ E6POS: X 774.0758, Y -19.4691, Z -124.0150, A 0, B 90, C 0, E1 0, E2 0, E3 0, E4 0 } C_DIS
LIN{ E6POS: X 773.1013, Y -19.2450, Z -124.0150, A 0, B 90, C 0, E1 0, E2 0, E3 0, E4 0 } C_DIS
LIN{ E6POS: X 772.1267, Y -19.0209, Z -124.0150, A 0, B 90, C 0, E1 0, E2 0, E3 0, E4 0 } C_DIS
LIN{ E6POS: X 771.1521, Y -18.7968, Z -124.0150, A 0, B 90, C 0, E1 0, E2 0, E3 0, E4 0 } C_DIS
LIN{ E6POS: X 770.3525, Y -18.6130, Z -124.0150, A 0, B 90, C 0, E1 0, E2 0, E3 0, E4 0 } C_DIS
LIN{ E6POS: X 770.3525, Y -18.6130, Z -124.0150, A 0, B 90, C 0, E1 0, E2 0, E3 0, E4 0 } C_DIS
LIN{ E6POS: X 769.3607, Y -18.4853, Z -124.0150, A 0, B 90, C 0, E1 0, E2 0, E3 0, E4 0 } C_DIS
LIN{ E6POS: X 768.3689, Y -18.3577, Z -124.0150, A 0, B 90, C 0, E1 0, E2 0, E3 0, E4 0 } C_DIS
LIN{ E6POS: X 767.3770, Y -18.2300, Z -124.0150, A 0, B 90, C 0, E1 0, E2 0, E3 0, E4 0 } C_DIS
LIN{ E6POS: X 766.3852, Y -18.1024, Z -124.0150, A 0, B 90, C 0, E1 0, E2 0, E3 0, E4 0 } C_DIS
LIN{ E6POS: X 765.3934, Y -17.9747, Z -124.0150, A 0, B 90, C 0, E1 0, E2 0, E3 0, E4 0 } C_DIS
LIN{ E6POS: X 764.4016, Y -17.8471, Z -124.0150, A 0, B 90, C 0, E1 0, E2 0, E3 0, E4 0 } C_DIS
LIN{ E6POS: X 763.4098, Y -17.7194, Z -124.0150, A 0, B 90, C 0, E1 0, E2 0, E3 0, E4 0 } C_DIS
LIN{ E6POS: X 762.4180, Y -17.5918, Z -124.0150, A 0, B 90, C 0, E1 0, E2 0, E3 0, E4 0 } C_DIS
LIN{ E6POS: X 762.3107, Y -17.5780, Z -124.0150, A 0, B 90, C 0, E1 0, E2 0, E3 0, E4 0 } C_DIS
LIN{ E6POS: X 762.3107, Y -17.5780, Z -124.0150, A 0, B 90, C 0, E1 0, E2 0, E3 0, E4 0 } C_DIS
LIN{ E6POS: X 761.3129, Y -17.5108, Z -124.0150, A 0, B 90, C 0, E1 0, E2 0, E3 0, E4 0 } C_DIS
LIN{ E6POS: X 760.3152, Y -17.4437, Z -124.0150, A 0, B 90, C 0, E1 0, E2 0, E3 0, E4 0 } C_DIS
LIN{ E6POS: X 759.3174, Y -17.3766, Z -124.0150, A 0, B 90, C 0, E1 0, E2 0, E3 0, E4 0 } C_DIS
LIN{ E6POS: X 758.3197, Y -17.3095, Z -124.0150, A 0, B 90, C 0, E1 0, E2 0, E3 0, E4 0 } C_DIS
LIN{ E6POS: X 757.3219, Y -17.2424, Z -124.0150, A 0, B 90, C 0, E1 0, E2 0, E3 0, E4 0 } C_DIS
LIN{ E6POS: X 756.3242, Y -17.1753, Z -124.0150, A 0, B 90, C 0, E1 0, E2 0, E3 0, E4 0 } C_DIS
LIN{ E6POS: X 755.3264, Y -17.1081, Z -124.0150, A 0, B 90, C 0, E1 0, E2 0, E3 0, E4 0 } C_DIS
LIN{ E6POS: X 754.3287, Y -17.0410, Z -124.0150, A 0, B 90, C 0, E1 0, E2 0, E3 0, E4 0 } C_DIS
LIN{ E6POS: X 753.8559, Y -17.0092, Z -124.0150, A 0, B 90, C 0, E1 0, E2 0, E3 0, E4 0 } C_DIS
LIN{ E6POS: X 753.8559, Y -17.0092, Z -124.0150, A 0, B 90, C 0, E1 0, E2 0, E3 0, E4 0 } C_DIS
LIN{ E6POS: X 752.8561, Y -16.9930, Z -124.0150, A 0, B 90, C 0, E1 0, E2 0, E3 0, E4 0 } C_DIS
LIN{ E6POS: X 751.8562, Y -16.9767, Z -124.0150, A 0, B 90, C 0, E1 0, E2 0, E3 0, E4 0 } C_DIS
LIN{ E6POS: X 750.8563, Y -16.9605, Z -124.0150, A 0, B 90, C 0, E1 0, E2 0, E3 0, E4 0 } C_DIS
LIN{ E6POS: X 749.8565, Y -16.9442, Z -124.0150, A 0, B 90, C 0, E1 0, E2 0, E3 0, E4 0 } C_DIS
LIN{ E6POS: X 748.8566, Y -16.9280, Z -124.0150, A 0, B 90, C 0, E1 0, E2 0, E3 0, E4 0 } C_DIS
LIN{ E6POS: X 747.8567, Y -16.9117, Z -124.0150, A 0, B 90, C 0, E1 0, E2 0, E3 0, E4 0 } C_DIS
LIN{ E6POS: X 746.8568, Y -16.8955, Z -124.0150, A 0, B 90, C 0, E1 0, E2 0, E3 0, E4 0 } C_DIS
LIN{ E6POS: X 745.9679, Y -16.8810, Z -124.0150, A 0, B 90, C 0, E1 0, E2 0, E3 0, E4 0 } C_DIS
LIN{ E6POS: X 745.9679, Y -16.8810, Z -124.0150, A 0, B 90, C 0, E1 0, E2 0, E3 0, E4 0 } C_DIS
LIN{ E6POS: X 744.9690, Y -16.9258, Z -124.0150, A 0, B 90, C 0, E1 0, E2 0, E3 0, E4 0 } C_DIS
LIN{ E6POS: X 743.9700, Y -16.9706, Z -124.0150, A 0, B 90, C 0, E1 0, E2 0, E3 0, E4 0 } C_DIS
LIN{ E6POS: X 742.9710, Y -17.0153, Z -124.0150, A 0, B 90, C 0, E1 0, E2 0, E3 0, E4 0 } C_DIS
LIN{ E6POS: X 741.9720, Y -17.0601, Z -124.0150, A 0, B 90, C 0, E1 0, E2 0, E3 0, E4 0 } C_DIS
LIN{ E6POS: X 740.9730, Y -17.1048, Z -124.0150, A 0, B 90, C 0, E1 0, E2 0, E3 0, E4 0 } C_DIS
LIN{ E6POS: X 739.9740, Y -17.1496, Z -124.0150, A 0, B 90, C 0, E1 0, E2 0, E3 0, E4 0 } C_DIS
LIN{ E6POS: X 739.6280, Y -17.1651, Z -124.0150, A 0, B 90, C 0, E1 0, E2 0, E3 0, E4 0 } C_DIS
LIN{ E6POS: X 739.6280, Y -17.1651, Z -124.0150, A 0, B 90, C 0, E1 0, E2 0, E3 0, E4 0 } C_DIS
LIN{ E6POS: X 738.6431, Y -17.3383, Z -124.0150, A 0, B 90, C 0, E1 0, E2 0, E3 0, E4 0 } C_DIS
LIN{ E6POS: X 737.6582, Y -17.5116, Z -124.0150, A 0, B 90, C 0, E1 0, E2 0, E3 0, E4 0 } C_DIS
LIN{ E6POS: X 736.6734, Y -17.6848, Z -124.0150, A 0, B 90, C 0, E1 0, E2 0, E3 0, E4 0 } C_DIS
LIN{ E6POS: X 735.8158, Y -17.8356, Z -124.0150, A 0, B 90, C 0, E1 0, E2 0, E3 0, E4 0 } C_DIS
LIN{ E6POS: X 735.8158, Y -17.8356, Z -124.0150, A 0, B 90, C 0, E1 0, E2 0, E3 0, E4 0 } C_DIS
LIN{ E6POS: X 735.0373, Y -18.4634, Z -124.0150, A 0, B 90, C 0, E1 0, E2 0, E3 0, E4 0 } C_DIS
LIN{ E6POS: X 734.5346, Y -18.8688, Z -124.0150, A 0, B 90, C 0, E1 0, E2 0, E3 0, E4 0 } C_DIS
LIN{ E6POS: X 735.2074, Y -19.6086, Z -124.0150, A 0, B 90, C 0, E1 0, E2 0, E3 0, E4 0 } C_DIS
LIN{ E6POS: X 735.7865, Y -20.2454, Z -124.0150, A 0, B 90, C 0, E1 0, E2 0, E3 0, E4 0 } C_DIS
LIN{ E6POS: X 735.7865, Y -20.2454, Z -124.0150, A 0, B 90, C 0, E1 0, E2 0, E3 0, E4 0 } C_DIS
LIN{ E6POS: X 736.6989, Y -20.6545, Z -124.0150, A 0, B 90, C 0, E1 0, E2 0, E3 0, E4 0 } C_DIS
LIN{ E6POS: X 737.6114, Y -21.0637, Z -124.0150, A 0, B 90, C 0, E1 0, E2 0, E3 0, E4 0 } C_DIS
LIN{ E6POS: X 738.5239, Y -21.4728, Z -124.0150, A 0, B 90, C 0, E1 0, E2 0, E3 0, E4 0 } C_DIS
LIN{ E6POS: X 739.4364, Y -21.8819, Z -124.0150, A 0, B 90, C 0, E1 0, E2 0, E3 0, E4 0 } C_DIS
LIN{ E6POS: X 739.5726, Y -21.9430, Z -124.0150, A 0, B 90, C 0, E1 0, E2 0, E3 0, E4 0 } C_DIS
LIN{ E6POS: X 739.5726, Y -21.9430, Z -124.0150, A 0, B 90, C 0, E1 0, E2 0, E3 0, E4 0 } C_DIS
LIN{ E6POS: X 740.5262, Y -22.2441, Z -124.0150, A 0, B 90, C 0, E1 0, E2 0, E3 0, E4 0 } C_DIS
LIN{ E6POS: X 741.4798, Y -22.5452, Z -124.0150, A 0, B 90, C 0, E1 0, E2 0, E3 0, E4 0 } C_DIS
LIN{ E6POS: X 742.4334, Y -22.8463, Z -124.0150, A 0, B 90, C 0, E1 0, E2 0, E3 0, E4 0 } C_DIS
LIN{ E6POS: X 743.3869, Y -23.1474, Z -124.0150, A 0, B 90, C 0, E1 0, E2 0, E3 0, E4 0 } C_DIS
LIN{ E6POS: X 744.3405, Y -23.4485, Z -124.0150, A 0, B 90, C 0, E1 0, E2 0, E3 0, E4 0 } C_DIS
LIN{ E6POS: X 745.2941, Y -23.7496, Z -124.0150, A 0, B 90, C 0, E1 0, E2 0, E3 0, E4 0 } C_DIS
LIN{ E6POS: X 745.8957, Y -23.9396, Z -124.0150, A 0, B 90, C 0, E1 0, E2 0, E3 0, E4 0 } C_DIS
LIN{ E6POS: X 745.8957, Y -23.9396, Z -124.0150, A 0, B 90, C 0, E1 0, E2 0, E3 0, E4 0 } C_DIS
LIN{ E6POS: X 746.8650, Y -24.1854, Z -124.0150, A 0, B 90, C 0, E1 0, E2 0, E3 0, E4 0 } C_DIS
LIN{ E6POS: X 747.8344, Y -24.4311, Z -124.0150, A 0, B 90, C 0, E1 0, E2 0, E3 0, E4 0 } C_DIS
LIN{ E6POS: X 748.8037, Y -24.6769, Z -124.0150, A 0, B 90, C 0, E1 0, E2 0, E3 0, E4 0 } C_DIS
LIN{ E6POS: X 749.7730, Y -24.9226, Z -124.0150, A 0, B 90, C 0, E1 0, E2 0, E3 0, E4 0 } C_DIS
LIN{ E6POS: X 750.7424, Y -25.1684, Z -124.0150, A 0, B 90, C 0, E1 0, E2 0, E3 0, E4 0 } C_DIS
LIN{ E6POS: X 751.7117, Y -25.4141, Z -124.0150, A 0, B 90, C 0, E1 0, E2 0, E3 0, E4 0 } C_DIS
LIN{ E6POS: X 752.6810, Y -25.6599, Z -124.0150, A 0, B 90, C 0, E1 0, E2 0, E3 0, E4 0 } C_DIS
LIN{ E6POS: X 753.6504, Y -25.9057, Z -124.0150, A 0, B 90, C 0, E1 0, E2 0, E3 0, E4 0 } C_DIS
LIN{ E6POS: X 753.7756, Y -25.9374, Z -124.0150, A 0, B 90, C 0, E1 0, E2 0, E3 0, E4 0 } C_DIS
LIN{ E6POS: X 753.7756, Y -25.9374, Z -124.0150, A 0, B 90, C 0, E1 0, E2 0, E3 0, E4 0 } C_DIS
LIN{ E6POS: X 754.7560, Y -26.1346, Z -124.0150, A 0, B 90, C 0, E1 0, E2 0, E3 0, E4 0 } C_DIS
LIN{ E6POS: X 755.7363, Y -26.3318, Z -124.0150, A 0, B 90, C 0, E1 0, E2 0, E3 0, E4 0 } C_DIS
LIN{ E6POS: X 756.7167, Y -26.5290, Z -124.0150, A 0, B 90, C 0, E1 0, E2 0, E3 0, E4 0 } C_DIS
LIN{ E6POS: X 757.6970, Y -26.7262, Z -124.0150, A 0, B 90, C 0, E1 0, E2 0, E3 0, E4 0 } C_DIS
LIN{ E6POS: X 758.6774, Y -26.9234, Z -124.0150, A 0, B 90, C 0, E1 0, E2 0, E3 0, E4 0 } C_DIS
LIN{ E6POS: X 759.6578, Y -27.1206, Z -124.0150, A 0, B 90, C 0, E1 0, E2 0, E3 0, E4 0 } C_DIS
LIN{ E6POS: X 760.6381, Y -27.3178, Z -124.0150, A 0, B 90, C 0, E1 0, E2 0, E3 0, E4 0 } C_DIS
LIN{ E6POS: X 761.6185, Y -27.5150, Z -124.0150, A 0, B 90, C 0, E1 0, E2 0, E3 0, E4 0 } C_DIS
LIN{ E6POS: X 762.2293, Y -27.6379, Z -124.0150, A 0, B 90, C 0, E1 0, E2 0, E3 0, E4 0 } C_DIS
LIN{ E6POS: X 762.2293, Y -27.6379, Z -124.0150, A 0, B 90, C 0, E1 0, E2 0, E3 0, E4 0 } C_DIS
LIN{ E6POS: X 763.2200, Y -27.7738, Z -124.0150, A 0, B 90, C 0, E1 0, E2 0, E3 0, E4 0 } C_DIS
LIN{ E6POS: X 764.2107, Y -27.9098, Z -124.0150, A 0, B 90, C 0, E1 0, E2 0, E3 0, E4 0 } C_DIS
LIN{ E6POS: X 765.2015, Y -28.0458, Z -124.0150, A 0, B 90, C 0, E1 0, E2 0, E3 0, E4 0 } C_DIS
LIN{ E6POS: X 766.1922, Y -28.1818, Z -124.0150, A 0, B 90, C 0, E1 0, E2 0, E3 0, E4 0 } C_DIS
LIN{ E6POS: X 767.1829, Y -28.3177, Z -124.0150, A 0, B 90, C 0, E1 0, E2 0, E3 0, E4 0 } C_DIS
LIN{ E6POS: X 768.1736, Y -28.4537, Z -124.0150, A 0, B 90, C 0, E1 0, E2 0, E3 0, E4 0 } C_DIS
LIN{ E6POS: X 769.1643, Y -28.5897, Z -124.0150, A 0, B 90, C 0, E1 0, E2 0, E3 0, E4 0 } C_DIS
LIN{ E6POS: X 770.1550, Y -28.7257, Z -124.0150, A 0, B 90, C 0, E1 0, E2 0, E3 0, E4 0 } C_DIS
LIN{ E6POS: X 770.2777, Y -28.7425, Z -124.0150, A 0, B 90, C 0, E1 0, E2 0, E3 0, E4 0 } C_DIS
LIN{ E6POS: X 770.2777, Y -28.7425, Z -124.0150, A 0, B 90, C 0, E1 0, E2 0, E3 0, E4 0 } C_DIS
LIN{ E6POS: X 771.2772, Y -28.7742, Z -124.0150, A 0, B 90, C 0, E1 0, E2 0, E3 0, E4 0 } C_DIS
LIN{ E6POS: X 772.2767, Y -28.8059, Z -124.0150, A 0, B 90, C 0, E1 0, E2 0, E3 0, E4 0 } C_DIS
LIN{ E6POS: X 773.2762, Y -28.8376, Z -124.0150, A 0, B 90, C 0, E1 0, E2 0, E3 0, E4 0 } C_DIS
LIN{ E6POS: X 774.2757, Y -28.8693, Z -124.0150, A 0, B 90, C 0, E1 0, E2 0, E3 0, E4 0 } C_DIS
LIN{ E6POS: X 775.2752, Y -28.9010, Z -124.0150, A 0, B 90, C 0, E1 0, E2 0, E3 0, E4 0 } C_DIS
LIN{ E6POS: X 776.2747, Y -28.9327, Z -124.0150, A 0, B 90, C 0, E1 0, E2 0, E3 0, E4 0 } C_DIS
LIN{ E6POS: X 776.9377, Y -28.9537, Z -124.0150, A 0, B 90, C 0, E1 0, E2 0, E3 0, E4 0 } C_DIS
LIN{ E6POS: X 776.9377, Y -28.9537, Z -124.0150, A 0, B 90, C 0, E1 0, E2 0, E3 0, E4 0 } C_DIS
LIN{ E6POS: X 777.9203, Y -29.1394, Z -124.0150, A 0, B 90, C 0, E1 0, E2 0, E3 0, E4 0 } C_DIS
LIN{ E6POS: X 778.9029, Y -29.3250, Z -124.0150, A 0, B 90, C 0, E1 0, E2 0, E3 0, E4 0 } C_DIS
LIN{ E6POS: X 779.8856, Y -29.5106, Z -124.0150, A 0, B 90, C 0, E1 0, E2 0, E3 0, E4 0 } C_DIS
LIN{ E6POS: X 780.8682, Y -29.6962, Z -124.0150, A 0, B 90, C 0, E1 0, E2 0, E3 0, E4 0 } C_DIS
LIN{ E6POS: X 781.8508, Y -29.8818, Z -124.0150, A 0, B 90, C 0, E1 0, E2 0, E3 0, E4 0 } C_DIS
LIN{ E6POS: X 781.9682, Y -29.9040, Z -124.0150, A 0, B 90, C 0, E1 0, E2 0, E3 0, E4 0 } C_DIS
LIN{ E6POS: X 781.9682, Y -29.9040, Z -124.0150, A 0, B 90, C 0, E1 0, E2 0, E3 0, E4 0 } C_DIS
LIN{ E6POS: X 782.6574, Y -30.6286, Z -124.0150, A 0, B 90, C 0, E1 0, E2 0, E3 0, E4 0 } C_DIS
LIN{ E6POS: X 783.3465, Y -31.3532, Z -124.0150, A 0, B 90, C 0, E1 0, E2 0, E3 0, E4 0 } C_DIS
LIN{ E6POS: X 784.0356, Y -32.0779, Z -124.0150, A 0, B 90, C 0, E1 0, E2 0, E3 0, E4 0 } C_DIS
LIN{ E6POS: X 784.7248, Y -32.8025, Z -124.0150, A 0, B 90, C 0, E1 0, E2 0, E3 0, E4 0 } C_DIS
LIN{ E6POS: X 785.1281, Y -33.2266, Z -124.0150, A 0, B 90, C 0, E1 0, E2 0, E3 0, E4 0 } C_DIS
LIN{ E6POS: X 785.1281, Y -33.2266, Z -124.0150, A 0, B 90, C 0, E1 0, E2 0, E3 0, E4 0 } C_DIS
LIN{ E6POS: X 785.2695, Y -34.2166, Z -124.0150, A 0, B 90, C 0, E1 0, E2 0, E3 0, E4 0 } C_DIS
LIN{ E6POS: X 785.4109, Y -35.2065, Z -124.0150, A 0, B 90, C 0, E1 0, E2 0, E3 0, E4 0 } C_DIS
LIN{ E6POS: X 785.5523, Y -36.1965, Z -124.0150, A 0, B 90, C 0, E1 0, E2 0, E3 0, E4 0 } C_DIS
LIN{ E6POS: X 785.6937, Y -37.1864, Z -124.0150, A 0, B 90, C 0, E1 0, E2 0, E3 0, E4 0 } C_DIS
LIN{ E6POS: X 785.8351, Y -38.1764, Z -124.0150, A 0, B 90, C 0, E1 0, E2 0, E3 0, E4 0 } C_DIS
LIN{ E6POS: X 785.9765, Y -39.1663, Z -124.0150, A 0, B 90, C 0, E1 0, E2 0, E3 0, E4 0 } C_DIS
LIN{ E6POS: X 786.1179, Y -40.1563, Z -124.0150, A 0, B 90, C 0, E1 0, E2 0, E3 0, E4 0 } C_DIS
LIN{ E6POS: X 786.1747, Y -40.5536, Z -124.0150, A 0, B 90, C 0, E1 0, E2 0, E3 0, E4 0 } C_DIS
LIN{ E6POS: X 786.1747, Y -40.5536, Z -124.0150, A 0, B 90, C 0, E1 0, E2 0, E3 0, E4 0 } C_DIS
LIN{ E6POS: X 786.0743, Y -41.5485, Z -124.0150, A 0, B 90, C 0, E1 0, E2 0, E3 0, E4 0 } C_DIS
LIN{ E6POS: X 785.9740, Y -42.5435, Z -124.0150, A 0, B 90, C 0, E1 0, E2 0, E3 0, E4 0 } C_DIS
LIN{ E6POS: X 785.8737, Y -43.5384, Z -124.0150, A 0, B 90, C 0, E1 0, E2 0, E3 0, E4 0 } C_DIS
LIN{ E6POS: X 785.7734, Y -44.5334, Z -124.0150, A 0, B 90, C 0, E1 0, E2 0, E3 0, E4 0 } C_DIS
LIN{ E6POS: X 785.6731, Y -45.5283, Z -124.0150, A 0, B 90, C 0, E1 0, E2 0, E3 0, E4 0 } C_DIS
LIN{ E6POS: X 785.5728, Y -46.5233, Z -124.0150, A 0, B 90, C 0, E1 0, E2 0, E3 0, E4 0 } C_DIS
LIN{ E6POS: X 785.4725, Y -47.5183, Z -124.0150, A 0, B 90, C 0, E1 0, E2 0, E3 0, E4 0 } C_DIS
LIN{ E6POS: X 785.3721, Y -48.5132, Z -124.0150, A 0, B 90, C 0, E1 0, E2 0, E3 0, E4 0 } C_DIS
LIN{ E6POS: X 785.2718, Y -49.5082, Z -124.0150, A 0, B 90, C 0, E1 0, E2 0, E3 0, E4 0 } C_DIS
LIN{ E6POS: X 785.1715, Y -50.5031, Z -124.0150, A 0, B 90, C 0, E1 0, E2 0, E3 0, E4 0 } C_DIS
LIN{ E6POS: X 785.0712, Y -51.4981, Z -124.0150, A 0, B 90, C 0, E1 0, E2 0, E3 0, E4 0 } C_DIS
LIN{ E6POS: X 784.9709, Y -52.4930, Z -124.0150, A 0, B 90, C 0, E1 0, E2 0, E3 0, E4 0 } C_DIS
LIN{ E6POS: X 784.8706, Y -53.4880, Z -124.0150, A 0, B 90, C 0, E1 0, E2 0, E3 0, E4 0 } C_DIS
LIN{ E6POS: X 784.8675, Y -53.5185, Z -124.0150, A 0, B 90, C 0, E1 0, E2 0, E3 0, E4 0 } C_DIS
LIN{ E6POS: X 784.8675, Y -53.5185, Z -124.0150, A 0, B 90, C 0, E1 0, E2 0, E3 0, E4 0 } C_DIS
LIN{ E6POS: X 784.6915, Y -54.5029, Z -124.0150, A 0, B 90, C 0, E1 0, E2 0, E3 0, E4 0 } C_DIS
LIN{ E6POS: X 784.5156, Y -55.4873, Z -124.0150, A 0, B 90, C 0, E1 0, E2 0, E3 0, E4 0 } C_DIS
LIN{ E6POS: X 784.3396, Y -56.4717, Z -124.0150, A 0, B 90, C 0, E1 0, E2 0, E3 0, E4 0 } C_DIS
LIN{ E6POS: X 784.1637, Y -57.4560, Z -124.0150, A 0, B 90, C 0, E1 0, E2 0, E3 0, E4 0 } C_DIS
LIN{ E6POS: X 783.9877, Y -58.4404, Z -124.0150, A 0, B 90, C 0, E1 0, E2 0, E3 0, E4 0 } C_DIS
LIN{ E6POS: X 783.8118, Y -59.4248, Z -124.0150, A 0, B 90, C 0, E1 0, E2 0, E3 0, E4 0 } C_DIS
LIN{ E6POS: X 783.6358, Y -60.4092, Z -124.0150, A 0, B 90, C 0, E1 0, E2 0, E3 0, E4 0 } C_DIS
LIN{ E6POS: X 783.4599, Y -61.3936, Z -124.0150, A 0, B 90, C 0, E1 0, E2 0, E3 0, E4 0 } C_DIS
LIN{ E6POS: X 783.2839, Y -62.3780, Z -124.0150, A 0, B 90, C 0, E1 0, E2 0, E3 0, E4 0 } C_DIS
LIN{ E6POS: X 783.1080, Y -63.3624, Z -124.0150, A 0, B 90, C 0, E1 0, E2 0, E3 0, E4 0 } C_DIS
LIN{ E6POS: X 782.9320, Y -64.3468, Z -124.0150, A 0, B 90, C 0, E1 0, E2 0, E3 0, E4 0 } C_DIS
LIN{ E6POS: X 782.7561, Y -65.3312, Z -124.0150, A 0, B 90, C 0, E1 0, E2 0, E3 0, E4 0 } C_DIS
LIN{ E6POS: X 782.5801, Y -66.3156, Z -124.0150, A 0, B 90, C 0, E1 0, E2 0, E3 0, E4 0 } C_DIS
LIN{ E6POS: X 782.4042, Y -67.3000, Z -124.0150, A 0, B 90, C 0, E1 0, E2 0, E3 0, E4 0 } C_DIS
LIN{ E6POS: X 782.2282, Y -68.2844, Z -124.0150, A 0, B 90, C 0, E1 0, E2 0, E3 0, E4 0 } C_DIS
LIN{ E6POS: X 782.0523, Y -69.2688, Z -124.0150, A 0, B 90, C 0, E1 0, E2 0, E3 0, E4 0 } C_DIS
LIN{ E6POS: X 781.8763, Y -70.2532, Z -124.0150, A 0, B 90, C 0, E1 0, E2 0, E3 0, E4 0 } C_DIS
LIN{ E6POS: X 781.7943, Y -70.7119, Z -124.0150, A 0, B 90, C 0, E1 0, E2 0, E3 0, E4 0 } C_DIS
LIN{ E6POS: X 781.7943, Y -70.7119, Z -124.0150, A 0, B 90, C 0, E1 0, E2 0, E3 0, E4 0 } C_DIS
LIN{ E6POS: X 781.5865, Y -71.6900, Z -124.0150, A 0, B 90, C 0, E1 0, E2 0, E3 0, E4 0 } C_DIS
LIN{ E6POS: X 781.3787, Y -72.6682, Z -124.0150, A 0, B 90, C 0, E1 0, E2 0, E3 0, E4 0 } C_DIS
LIN{ E6POS: X 781.1709, Y -73.6464, Z -124.0150, A 0, B 90, C 0, E1 0, E2 0, E3 0, E4 0 } C_DIS
LIN{ E6POS: X 780.9631, Y -74.6245, Z -124.0150, A 0, B 90, C 0, E1 0, E2 0, E3 0, E4 0 } C_DIS
LIN{ E6POS: X 780.7553, Y -75.6027, Z -124.0150, A 0, B 90, C 0, E1 0, E2 0, E3 0, E4 0 } C_DIS
LIN{ E6POS: X 780.5475, Y -76.5809, Z -124.0150, A 0, B 90, C 0, E1 0, E2 0, E3 0, E4 0 } C_DIS
LIN{ E6POS: X 780.3397, Y -77.5590, Z -124.0150, A 0, B 90, C 0, E1 0, E2 0, E3 0, E4 0 } C_DIS
LIN{ E6POS: X 780.1319, Y -78.5372, Z -124.0150, A 0, B 90, C 0, E1 0, E2 0, E3 0, E4 0 } C_DIS
LIN{ E6POS: X 779.9241, Y -79.5154, Z -124.0150, A 0, B 90, C 0, E1 0, E2 0, E3 0, E4 0 } C_DIS
LIN{ E6POS: X 779.7163, Y -80.4936, Z -124.0150, A 0, B 90, C 0, E1 0, E2 0, E3 0, E4 0 } C_DIS
LIN{ E6POS: X 779.5085, Y -81.4717, Z -124.0150, A 0, B 90, C 0, E1 0, E2 0, E3 0, E4 0 } C_DIS
LIN{ E6POS: X 779.3007, Y -82.4499, Z -124.0150, A 0, B 90, C 0, E1 0, E2 0, E3 0, E4 0 } C_DIS
LIN{ E6POS: X 779.0929, Y -83.4281, Z -124.0150, A 0, B 90, C 0, E1 0, E2 0, E3 0, E4 0 } C_DIS
LIN{ E6POS: X 778.8851, Y -84.4062, Z -124.0150, A 0, B 90, C 0, E1 0, E2 0, E3 0, E4 0 } C_DIS
LIN{ E6POS: X 778.6773, Y -85.3844, Z -124.0150, A 0, B 90, C 0, E1 0, E2 0, E3 0, E4 0 } C_DIS
LIN{ E6POS: X 778.4695, Y -86.3626, Z -124.0150, A 0, B 90, C 0, E1 0, E2 0, E3 0, E4 0 } C_DIS
LIN{ E6POS: X 778.2617, Y -87.3408, Z -124.0150, A 0, B 90, C 0, E1 0, E2 0, E3 0, E4 0 } C_DIS
LIN{ E6POS: X 778.0539, Y -88.3189, Z -124.0150, A 0, B 90, C 0, E1 0, E2 0, E3 0, E4 0 } C_DIS
LIN{ E6POS: X 777.8461, Y -89.2971, Z -124.0150, A 0, B 90, C 0, E1 0, E2 0, E3 0, E4 0 } C_DIS
LIN{ E6POS: X 777.6383, Y -90.2753, Z -124.0150, A 0, B 90, C 0, E1 0, E2 0, E3 0, E4 0 } C_DIS
LIN{ E6POS: X 777.5429, Y -90.7243, Z -124.0150, A 0, B 90, C 0, E1 0, E2 0, E3 0, E4 0 } C_DIS
LIN{ E6POS: X 777.5429, Y -90.7243, Z -124.0150, A 0, B 90, C 0, E1 0, E2 0, E3 0, E4 0 } C_DIS
LIN{ E6POS: X 777.3226, Y -91.6997, Z -124.0150, A 0, B 90, C 0, E1 0, E2 0, E3 0, E4 0 } C_DIS
LIN{ E6POS: X 777.1022, Y -92.6751, Z -124.0150, A 0, B 90, C 0, E1 0, E2 0, E3 0, E4 0 } C_DIS
LIN{ E6POS: X 776.8819, Y -93.6506, Z -124.0150, A 0, B 90, C 0, E1 0, E2 0, E3 0, E4 0 } C_DIS
LIN{ E6POS: X 776.6615, Y -94.6260, Z -124.0150, A 0, B 90, C 0, E1 0, E2 0, E3 0, E4 0 } C_DIS
LIN{ E6POS: X 776.4412, Y -95.6014, Z -124.0150, A 0, B 90, C 0, E1 0, E2 0, E3 0, E4 0 } C_DIS
LIN{ E6POS: X 776.2208, Y -96.5768, Z -124.0150, A 0, B 90, C 0, E1 0, E2 0, E3 0, E4 0 } C_DIS
LIN{ E6POS: X 776.0005, Y -97.5522, Z -124.0150, A 0, B 90, C 0, E1 0, E2 0, E3 0, E4 0 } C_DIS
LIN{ E6POS: X 775.7802, Y -98.5277, Z -124.0150, A 0, B 90, C 0, E1 0, E2 0, E3 0, E4 0 } C_DIS
LIN{ E6POS: X 775.5598, Y -99.5031, Z -124.0150, A 0, B 90, C 0, E1 0, E2 0, E3 0, E4 0 } C_DIS
LIN{ E6POS: X 775.3395, Y -100.4785, Z -124.0150, A 0, B 90, C 0, E1 0, E2 0, E3 0, E4 0 } C_DIS
LIN{ E6POS: X 775.1191, Y -101.4539, Z -124.0150, A 0, B 90, C 0, E1 0, E2 0, E3 0, E4 0 } C_DIS
LIN{ E6POS: X 774.8988, Y -102.4294, Z -124.0150, A 0, B 90, C 0, E1 0, E2 0, E3 0, E4 0 } C_DIS
LIN{ E6POS: X 774.6784, Y -103.4048, Z -124.0150, A 0, B 90, C 0, E1 0, E2 0, E3 0, E4 0 } C_DIS
LIN{ E6POS: X 774.4581, Y -104.3802, Z -124.0150, A 0, B 90, C 0, E1 0, E2 0, E3 0, E4 0 } C_DIS
LIN{ E6POS: X 774.2377, Y -105.3556, Z -124.0150, A 0, B 90, C 0, E1 0, E2 0, E3 0, E4 0 } C_DIS
LIN{ E6POS: X 774.0174, Y -106.3310, Z -124.0150, A 0, B 90, C 0, E1 0, E2 0, E3 0, E4 0 } C_DIS
LIN{ E6POS: X 773.7970, Y -107.3065, Z -124.0150, A 0, B 90, C 0, E1 0, E2 0, E3 0, E4 0 } C_DIS
LIN{ E6POS: X 773.5767, Y -108.2819, Z -124.0150, A 0, B 90, C 0, E1 0, E2 0, E3 0, E4 0 } C_DIS
LIN{ E6POS: X 773.3564, Y -109.2573, Z -124.0150, A 0, B 90, C 0, E1 0, E2 0, E3 0, E4 0 } C_DIS
LIN{ E6POS: X 773.1360, Y -110.2327, Z -124.0150, A 0, B 90, C 0, E1 0, E2 0, E3 0, E4 0 } C_DIS
LIN{ E6POS: X 772.9157, Y -111.2082, Z -124.0150, A 0, B 90, C 0, E1 0, E2 0, E3 0, E4 0 } C_DIS
LIN{ E6POS: X 772.7038, Y -112.1462, Z -124.0150, A 0, B 90, C 0, E1 0, E2 0, E3 0, E4 0 } C_DIS
LIN{ E6POS: X 772.7038, Y -112.1462, Z -124.0150, A 0, B 90, C 0, E1 0, E2 0, E3 0, E4 0 } C_DIS
LIN{ E6POS: X 772.0412, Y -111.3972, Z -124.0150, A 0, B 90, C 0, E1 0, E2 0, E3 0, E4 0 } C_DIS
LIN{ E6POS: X 771.3787, Y -110.6481, Z -124.0150, A 0, B 90, C 0, E1 0, E2 0, E3 0, E4 0 } C_DIS
LIN{ E6POS: X 770.7162, Y -109.8991, Z -124.0150, A 0, B 90, C 0, E1 0, E2 0, E3 0, E4 0 } C_DIS
LIN{ E6POS: X 770.0537, Y -109.1500, Z -124.0150, A 0, B 90, C 0, E1 0, E2 0, E3 0, E4 0 } C_DIS
LIN{ E6POS: X 770.0315, Y -109.1250, Z -124.0150, A 0, B 90, C 0, E1 0, E2 0, E3 0, E4 0 } C_DIS
LIN{ E6POS: X 770.0315, Y -109.1250, Z -124.0150, A 0, B 90, C 0, E1 0, E2 0, E3 0, E4 0 } C_DIS
LIN{ E6POS: X 769.2905, Y -108.4535, Z -124.0150, A 0, B 90, C 0, E1 0, E2 0, E3 0, E4 0 } C_DIS
LIN{ E6POS: X 768.5495, Y -107.7819, Z -124.0150, A 0, B 90, C 0, E1 0, E2 0, E3 0, E4 0 } C_DIS
LIN{ E6POS: X 767.8086, Y -107.1104, Z -124.0150, A 0, B 90, C 0, E1 0, E2 0, E3 0, E4 0 } C_DIS
LIN{ E6POS: X 767.0676, Y -106.4389, Z -124.0150, A 0, B 90, C 0, E1 0, E2 0, E3 0, E4 0 } C_DIS
LIN{ E6POS: X 766.5551, Y -105.9745, Z -124.0150, A 0, B 90, C 0, E1 0, E2 0, E3 0, E4 0 } C_DIS
LIN{ E6POS: X 766.5551, Y -105.9745, Z -124.0150, A 0, B 90, C 0, E1 0, E2 0, E3 0, E4 0 } C_DIS
LIN{ E6POS: X 766.5551, Y -105.9745, Z -124.0150, A 0, B 90, C 0, E1 0, E2 0, E3 0, E4 0 } C_DIS
LIN{ E6POS: X 765.7244, Y -105.4178, Z -124.0150, A 0, B 90, C 0, E1 0, E2 0, E3 0, E4 0 } C_DIS
LIN{ E6POS: X 764.8937, Y -104.8610, Z -124.0150, A 0, B 90, C 0, E1 0, E2 0, E3 0, E4 0 } C_DIS
LIN{ E6POS: X 764.0630, Y -104.3043, Z -124.0150, A 0, B 90, C 0, E1 0, E2 0, E3 0, E4 0 } C_DIS
LIN{ E6POS: X 763.2323, Y -103.7476, Z -124.0150, A 0, B 90, C 0, E1 0, E2 0, E3 0, E4 0 } C_DIS
LIN{ E6POS: X 762.4016, Y -103.1909, Z -124.0150, A 0, B 90, C 0, E1 0, E2 0, E3 0, E4 0 } C_DIS
LIN{ E6POS: X 761.5709, Y -102.6341, Z -124.0150, A 0, B 90, C 0, E1 0, E2 0, E3 0, E4 0 } C_DIS
LIN{ E6POS: X 761.4725, Y -102.5682, Z -124.0150, A 0, B 90, C 0, E1 0, E2 0, E3 0, E4 0 } C_DIS
LIN{ E6POS: X 761.4725, Y -102.5682, Z -124.0150, A 0, B 90, C 0, E1 0, E2 0, E3 0, E4 0 } C_DIS
LIN{ E6POS: X 760.5803, Y -102.1166, Z -124.0150, A 0, B 90, C 0, E1 0, E2 0, E3 0, E4 0 } C_DIS
LIN{ E6POS: X 759.6881, Y -101.6650, Z -124.0150, A 0, B 90, C 0, E1 0, E2 0, E3 0, E4 0 } C_DIS
LIN{ E6POS: X 758.7958, Y -101.2135, Z -124.0150, A 0, B 90, C 0, E1 0, E2 0, E3 0, E4 0 } C_DIS
LIN{ E6POS: X 757.9036, Y -100.7619, Z -124.0150, A 0, B 90, C 0, E1 0, E2 0, E3 0, E4 0 } C_DIS
LIN{ E6POS: X 757.0114, Y -100.3103, Z -124.0150, A 0, B 90, C 0, E1 0, E2 0, E3 0, E4 0 } C_DIS
LIN{ E6POS: X 756.1191, Y -99.8587, Z -124.0150, A 0, B 90, C 0, E1 0, E2 0, E3 0, E4 0 } C_DIS
LIN{ E6POS: X 755.2269, Y -99.4072, Z -124.0150, A 0, B 90, C 0, E1 0, E2 0, E3 0, E4 0 } C_DIS
LIN{ E6POS: X 754.3347, Y -98.9556, Z -124.0150, A 0, B 90, C 0, E1 0, E2 0, E3 0, E4 0 } C_DIS
LIN{ E6POS: X 753.9790, Y -98.7756, Z -124.0150, A 0, B 90, C 0, E1 0, E2 0, E3 0, E4 0 } C_DIS
LIN{ E6POS: X 753.9790, Y -98.7756, Z -124.0150, A 0, B 90, C 0, E1 0, E2 0, E3 0, E4 0 } C_DIS
LIN{ E6POS: X 753.0513, Y -98.4023, Z -124.0150, A 0, B 90, C 0, E1 0, E2 0, E3 0, E4 0 } C_DIS
LIN{ E6POS: X 752.1235, Y -98.0291, Z -124.0150, A 0, B 90, C 0, E1 0, E2 0, E3 0, E4 0 } C_DIS
LIN{ E6POS: X 751.1958, Y -97.6558, Z -124.0150, A 0, B 90, C 0, E1 0, E2 0, E3 0, E4 0 } C_DIS
LIN{ E6POS: X 750.2681, Y -97.2826, Z -124.0150, A 0, B 90, C 0, E1 0, E2 0, E3 0, E4 0 } C_DIS
LIN{ E6POS: X 749.3403, Y -96.9094, Z -124.0150, A 0, B 90, C 0, E1 0, E2 0, E3 0, E4 0 } C_DIS
LIN{ E6POS: X 748.4126, Y -96.5361, Z -124.0150, A 0, B 90, C 0, E1 0, E2 0, E3 0, E4 0 } C_DIS
LIN{ E6POS: X 747.4849, Y -96.1629, Z -124.0150, A 0, B 90, C 0, E1 0, E2 0, E3 0, E4 0 } C_DIS
LIN{ E6POS: X 746.5571, Y -95.7896, Z -124.0150, A 0, B 90, C 0, E1 0, E2 0, E3 0, E4 0 } C_DIS
LIN{ E6POS: X 745.6294, Y -95.4164, Z -124.0150, A 0, B 90, C 0, E1 0, E2 0, E3 0, E4 0 } C_DIS
LIN{ E6POS: X 744.7017, Y -95.0431, Z -124.0150, A 0, B 90, C 0, E1 0, E2 0, E3 0, E4 0 } C_DIS
LIN{ E6POS: X 743.7739, Y -94.6699, Z -124.0150, A 0, B 90, C 0, E1 0, E2 0, E3 0, E4 0 } C_DIS
LIN{ E6POS: X 743.2721, Y -94.4680, Z -124.0150, A 0, B 90, C 0, E1 0, E2 0, E3 0, E4 0 } C_DIS
LIN{ E6POS: X 743.2721, Y -94.4680, Z -124.0150, A 0, B 90, C 0, E1 0, E2 0, E3 0, E4 0 } C_DIS
LIN{ E6POS: X 742.3318, Y -94.1277, Z -124.0150, A 0, B 90, C 0, E1 0, E2 0, E3 0, E4 0 } C_DIS
LIN{ E6POS: X 741.3914, Y -93.7875, Z -124.0150, A 0, B 90, C 0, E1 0, E2 0, E3 0, E4 0 } C_DIS
LIN{ E6POS: X 740.4511, Y -93.4472, Z -124.0150, A 0, B 90, C 0, E1 0, E2 0, E3 0, E4 0 } C_DIS
LIN{ E6POS: X 739.5108, Y -93.1069, Z -124.0150, A 0, B 90, C 0, E1 0, E2 0, E3 0, E4 0 } C_DIS
LIN{ E6POS: X 738.5704, Y -92.7667, Z -124.0150, A 0, B 90, C 0, E1 0, E2 0, E3 0, E4 0 } C_DIS
LIN{ E6POS: X 737.6301, Y -92.4264, Z -124.0150, A 0, B 90, C 0, E1 0, E2 0, E3 0, E4 0 } C_DIS
LIN{ E6POS: X 736.6898, Y -92.0862, Z -124.0150, A 0, B 90, C 0, E1 0, E2 0, E3 0, E4 0 } C_DIS
LIN{ E6POS: X 735.7494, Y -91.7459, Z -124.0150, A 0, B 90, C 0, E1 0, E2 0, E3 0, E4 0 } C_DIS
LIN{ E6POS: X 734.8091, Y -91.4057, Z -124.0150, A 0, B 90, C 0, E1 0, E2 0, E3 0, E4 0 } C_DIS
LIN{ E6POS: X 733.8688, Y -91.0654, Z -124.0150, A 0, B 90, C 0, E1 0, E2 0, E3 0, E4 0 } C_DIS
LIN{ E6POS: X 732.9284, Y -90.7252, Z -124.0150, A 0, B 90, C 0, E1 0, E2 0, E3 0, E4 0 } C_DIS
LIN{ E6POS: X 731.9881, Y -90.3849, Z -124.0150, A 0, B 90, C 0, E1 0, E2 0, E3 0, E4 0 } C_DIS
LIN{ E6POS: X 731.1327, Y -90.0754, Z -124.0150, A 0, B 90, C 0, E1 0, E2 0, E3 0, E4 0 } C_DIS
LIN{ E6POS: X 731.1327, Y -90.0754, Z -124.0150, A 0, B 90, C 0, E1 0, E2 0, E3 0, E4 0 } C_DIS
LIN{ E6POS: X 730.1869, Y -89.7505, Z -124.0150, A 0, B 90, C 0, E1 0, E2 0, E3 0, E4 0 } C_DIS
LIN{ E6POS: X 729.2412, Y -89.4256, Z -124.0150, A 0, B 90, C 0, E1 0, E2 0, E3 0, E4 0 } C_DIS
LIN{ E6POS: X 728.2954, Y -89.1007, Z -124.0150, A 0, B 90, C 0, E1 0, E2 0, E3 0, E4 0 } C_DIS
LIN{ E6POS: X 727.3497, Y -88.7758, Z -124.0150, A 0, B 90, C 0, E1 0, E2 0, E3 0, E4 0 } C_DIS
LIN{ E6POS: X 726.4040, Y -88.4509, Z -124.0150, A 0, B 90, C 0, E1 0, E2 0, E3 0, E4 0 } C_DIS
LIN{ E6POS: X 725.4582, Y -88.1260, Z -124.0150, A 0, B 90, C 0, E1 0, E2 0, E3 0, E4 0 } C_DIS
LIN{ E6POS: X 724.5125, Y -87.8011, Z -124.0150, A 0, B 90, C 0, E1 0, E2 0, E3 0, E4 0 } C_DIS
LIN{ E6POS: X 723.5667, Y -87.4762, Z -124.0150, A 0, B 90, C 0, E1 0, E2 0, E3 0, E4 0 } C_DIS
LIN{ E6POS: X 722.6210, Y -87.1513, Z -124.0150, A 0, B 90, C 0, E1 0, E2 0, E3 0, E4 0 } C_DIS
LIN{ E6POS: X 721.6752, Y -86.8264, Z -124.0150, A 0, B 90, C 0, E1 0, E2 0, E3 0, E4 0 } C_DIS
LIN{ E6POS: X 720.7295, Y -86.5015, Z -124.0150, A 0, B 90, C 0, E1 0, E2 0, E3 0, E4 0 } C_DIS
LIN{ E6POS: X 719.7837, Y -86.1766, Z -124.0150, A 0, B 90, C 0, E1 0, E2 0, E3 0, E4 0 } C_DIS
LIN{ E6POS: X 719.3423, Y -86.0250, Z -124.0150, A 0, B 90, C 0, E1 0, E2 0, E3 0, E4 0 } C_DIS
LIN{ E6POS: X 719.3423, Y -86.0250, Z -124.0150, A 0, B 90, C 0, E1 0, E2 0, E3 0, E4 0 } C_DIS
LIN{ E6POS: X 718.3954, Y -85.7035, Z -124.0150, A 0, B 90, C 0, E1 0, E2 0, E3 0, E4 0 } C_DIS
LIN{ E6POS: X 717.4485, Y -85.3819, Z -124.0150, A 0, B 90, C 0, E1 0, E2 0, E3 0, E4 0 } C_DIS
LIN{ E6POS: X 716.5016, Y -85.0604, Z -124.0150, A 0, B 90, C 0, E1 0, E2 0, E3 0, E4 0 } C_DIS
LIN{ E6POS: X 715.5547, Y -84.7389, Z -124.0150, A 0, B 90, C 0, E1 0, E2 0, E3 0, E4 0 } C_DIS
LIN{ E6POS: X 714.6078, Y -84.4174, Z -124.0150, A 0, B 90, C 0, E1 0, E2 0, E3 0, E4 0 } C_DIS
LIN{ E6POS: X 713.6609, Y -84.0958, Z -124.0150, A 0, B 90, C 0, E1 0, E2 0, E3 0, E4 0 } C_DIS
LIN{ E6POS: X 712.7140, Y -83.7743, Z -124.0150, A 0, B 90, C 0, E1 0, E2 0, E3 0, E4 0 } C_DIS
LIN{ E6POS: X 711.7671, Y -83.4528, Z -124.0150, A 0, B 90, C 0, E1 0, E2 0, E3 0, E4 0 } C_DIS
LIN{ E6POS: X 710.8202, Y -83.1313, Z -124.0150, A 0, B 90, C 0, E1 0, E2 0, E3 0, E4 0 } C_DIS
LIN{ E6POS: X 709.8733, Y -82.8097, Z -124.0150, A 0, B 90, C 0, E1 0, E2 0, E3 0, E4 0 } C_DIS
LIN{ E6POS: X 709.6832, Y -82.7452, Z -124.0150, A 0, B 90, C 0, E1 0, E2 0, E3 0, E4 0 } C_DIS
LIN{ E6POS: X 709.6832, Y -82.7452, Z -124.0150, A 0, B 90, C 0, E1 0, E2 0, E3 0, E4 0 } C_DIS
LIN{ E6POS: X 708.7429, Y -82.4049, Z -124.0150, A 0, B 90, C 0, E1 0, E2 0, E3 0, E4 0 } C_DIS
LIN{ E6POS: X 707.8026, Y -82.0645, Z -124.0150, A 0, B 90, C 0, E1 0, E2 0, E3 0, E4 0 } C_DIS
LIN{ E6POS: X 706.8623, Y -81.7242, Z -124.0150, A 0, B 90, C 0, E1 0, E2 0, E3 0, E4 0 } C_DIS
LIN{ E6POS: X 705.9220, Y -81.3838, Z -124.0150, A 0, B 90, C 0, E1 0, E2 0, E3 0, E4 0 } C_DIS
LIN{ E6POS: X 704.9817, Y -81.0435, Z -124.0150, A 0, B 90, C 0, E1 0, E2 0, E3 0, E4 0 } C_DIS
LIN{ E6POS: X 704.0414, Y -80.7032, Z -124.0150, A 0, B 90, C 0, E1 0, E2 0, E3 0, E4 0 } C_DIS
LIN{ E6POS: X 703.9355, Y -80.6648, Z -124.0150, A 0, B 90, C 0, E1 0, E2 0, E3 0, E4 0 } C_DIS
LIN{ E6POS: X 703.9355, Y -80.6648, Z -124.0150, A 0, B 90, C 0, E1 0, E2 0, E3 0, E4 0 } C_DIS
LIN{ E6POS: X 703.0134, Y -80.2779, Z -124.0150, A 0, B 90, C 0, E1 0, E2 0, E3 0, E4 0 } C_DIS
LIN{ E6POS: X 702.0913, Y -79.8909, Z -124.0150, A 0, B 90, C 0, E1 0, E2 0, E3 0, E4 0 } C_DIS
LIN{ E6POS: X 701.1692, Y -79.5039, Z -124.0150, A 0, B 90, C 0, E1 0, E2 0, E3 0, E4 0 } C_DIS
LIN{ E6POS: X 701.1214, Y -79.4838, Z -124.0150, A 0, B 90, C 0, E1 0, E2 0, E3 0, E4 0 } C_DIS
LIN{ E6POS: X 701.1214, Y -79.4838, Z -124.0150, A 0, B 90, C 0, E1 0, E2 0, E3 0, E4 0 } C_DIS
LIN{ E6POS: X 700.4111, Y -78.7799, Z -124.0150, A 0, B 90, C 0, E1 0, E2 0, E3 0, E4 0 } C_DIS
LIN{ E6POS: X 700.3453, Y -78.7147, Z -124.0150, A 0, B 90, C 0, E1 0, E2 0, E3 0, E4 0 } C_DIS
LIN{ E6POS: X 700.5830, Y -77.7433, Z -124.0150, A 0, B 90, C 0, E1 0, E2 0, E3 0, E4 0 } C_DIS
LIN{ E6POS: X 700.7129, Y -77.2124, Z -124.0150, A 0, B 90, C 0, E1 0, E2 0, E3 0, E4 0 } C_DIS
LIN{ E6POS: X 700.7129, Y -77.2124, Z -124.0150, A 0, B 90, C 0, E1 0, E2 0, E3 0, E4 0 } C_DIS
LIN{ E6POS: X 700.9430, Y -76.2392, Z -124.0150, A 0, B 90, C 0, E1 0, E2 0, E3 0, E4 0 } C_DIS
LIN{ E6POS: X 701.0454, Y -75.8061, Z -124.0150, A 0, B 90, C 0, E1 0, E2 0, E3 0, E4 0 } C_DIS
LIN{ E6POS: X 701.0454, Y -75.8061, Z -124.0150, A 0, B 90, C 0, E1 0, E2 0, E3 0, E4 0 } C_DIS
LIN{ E6POS: X 701.2811, Y -74.8343, Z -124.0150, A 0, B 90, C 0, E1 0, E2 0, E3 0, E4 0 } C_DIS
LIN{ E6POS: X 701.3851, Y -74.4053, Z -124.0150, A 0, B 90, C 0, E1 0, E2 0, E3 0, E4 0 } C_DIS
LIN{ E6POS: X 701.3851, Y -74.4053, Z -124.0150, A 0, B 90, C 0, E1 0, E2 0, E3 0, E4 0 } C_DIS
LIN{ E6POS: X 701.6299, Y -73.4357, Z -124.0150, A 0, B 90, C 0, E1 0, E2 0, E3 0, E4 0 } C_DIS
LIN{ E6POS: X 701.7366, Y -73.0133, Z -124.0150, A 0, B 90, C 0, E1 0, E2 0, E3 0, E4 0 } C_DIS
LIN{ E6POS: X 701.7366, Y -73.0133, Z -124.0150, A 0, B 90, C 0, E1 0, E2 0, E3 0, E4 0 } C_DIS
LIN{ E6POS: X 701.9925, Y -72.0466, Z -124.0150, A 0, B 90, C 0, E1 0, E2 0, E3 0, E4 0 } C_DIS
LIN{ E6POS: X 702.1028, Y -71.6301, Z -124.0150, A 0, B 90, C 0, E1 0, E2 0, E3 0, E4 0 } C_DIS
LIN{ E6POS: X 702.1028, Y -71.6301, Z -124.0150, A 0, B 90, C 0, E1 0, E2 0, E3 0, E4 0 } C_DIS
LIN{ E6POS: X 702.3630, Y -70.6645, Z -124.0150, A 0, B 90, C 0, E1 0, E2 0, E3 0, E4 0 } C_DIS
LIN{ E6POS: X 702.4768, Y -70.2420, Z -124.0150, A 0, B 90, C 0, E1 0, E2 0, E3 0, E4 0 } C_DIS
LIN{ E6POS: X 702.4768, Y -70.2420, Z -124.0150, A 0, B 90, C 0, E1 0, E2 0, E3 0, E4 0 } C_DIS
LIN{ E6POS: X 702.7332, Y -69.2754, Z -124.0150, A 0, B 90, C 0, E1 0, E2 0, E3 0, E4 0 } C_DIS
LIN{ E6POS: X 702.8503, Y -68.8341, Z -124.0150, A 0, B 90, C 0, E1 0, E2 0, E3 0, E4 0 } C_DIS
LIN{ E6POS: X 702.8503, Y -68.8341, Z -124.0150, A 0, B 90, C 0, E1 0, E2 0, E3 0, E4 0 } C_DIS
LIN{ E6POS: X 703.0953, Y -67.8645, Z -124.0150, A 0, B 90, C 0, E1 0, E2 0, E3 0, E4 0 } C_DIS
LIN{ E6POS: X 703.2152, Y -67.3901, Z -124.0150, A 0, B 90, C 0, E1 0, E2 0, E3 0, E4 0 } C_DIS
